LIN {X 0,Y 573.858,Z 220.468,A -85,B 0,C 180,E1 -2228.443,E2 -2228.443} C_VEL
LIN {X 0,Y 573.667,Z 239.844,A -85,B 0,C 180,E1 -2231.425,E2 -2231.425} C_VEL
LIN {X 0,Y 573.432,Z 259.15,A -85,B 0,C 180,E1 -2234.357,E2 -2234.357} C_VEL
LIN {X 0,Y 573.37,Z 271.275,A -85,B 0,C 180,E1 -2236.148,E2 -2236.148} C_VEL
LIN {X 0,Y 574.08,Z 276.429,A -85,B 0,C 180,E1 -2236.256,E2 -2236.256} C_VEL
LIN {X 0,Y 573.913,Z 378.895,A -85,B 0,C 180,E1 -2237.557,E2 -2237.557} C_VEL
LIN {X 0,Y 573.795,Z 392.184,A -85,B 0,C 180,E1 -2237.869,E2 -2237.869} C_VEL
LIN {X 0,Y 573.682,Z 404.351,A -85,B 0,C 180,E1 -2238.293,E2 -2238.293} C_VEL
LIN {X 0,Y 573.582,Z 416.727,A -85,B 0,C 180,E1 -2238.879,E2 -2238.879} C_VEL
LIN {X 0,Y 573.432,Z 428.185,A -85,B 0,C 180,E1 -2239.584,E2 -2239.584} C_VEL
LIN {X 0,Y 573.329,Z 438.59,A -85,B 0,C 180,E1 -2240.384,E2 -2240.384} C_VEL
LIN {X 0,Y 573.238,Z 447.066,A -85,B 0,C 180,E1 -2241.184,E2 -2241.184} C_VEL
LIN {X 0,Y 573.162,Z 454.952,A -85,B 0,C 180,E1 -2242.07,E2 -2242.07} C_VEL
LIN {X 0,Y 573.077,Z 462.942,A -85,B 0,C 180,E1 -2243.183,E2 -2243.183} C_VEL
LIN {X 0,Y 573.071,Z 469.674,A -85,B 0,C 180,E1 -2244.369,E2 -2244.369} C_VEL
LIN {X 0,Y 573.029,Z 474.368,A -85,B 0,C 180,E1 -2245.426,E2 -2245.426} C_VEL
LIN {X 0,Y 573.023,Z 477.954,A -85,B 0,C 180,E1 -2246.483,E2 -2246.483} C_VEL
LIN {X 0,Y 572.959,Z 479.805,A -85,B 0,C 180,E1 -2247.187,E2 -2247.187} C_VEL
LIN {X 0,Y 572.946,Z 482.184,A -85,B 0,C 180,E1 -2248.593,E2 -2248.593} C_VEL
LIN {X 0,Y 572.938,Z 483,A -85,B 0,C 180,E1 -2249.999,E2 -2249.999} C_VEL
LIN {X 0,Y 572.946,Z 482.187,A -85,B 0,C 180,E1 -2251.405,E2 -2251.405} C_VEL
LIN {X 0,Y 572.959,Z 479.813,A -85,B 0,C 180,E1 -2252.811,E2 -2252.811} C_VEL
LIN {X 0,Y 573.014,Z 476.899,A -85,B 0,C 180,E1 -2253.867,E2 -2253.867} C_VEL
LIN {X 0,Y 572.963,Z 472.953,A -85,B 0,C 180,E1 -2254.924,E2 -2254.924} C_VEL
LIN {X 0,Y 573.093,Z 467.873,A -85,B 0,C 180,E1 -2255.982,E2 -2255.982} C_VEL
LIN {X 0,Y 573.083,Z 461.476,A -85,B 0,C 180,E1 -2257.043,E2 -2257.043} C_VEL
LIN {X 0,Y 573.175,Z 453.488,A -85,B 0,C 180,E1 -2258.105,E2 -2258.105} C_VEL
LIN {X 0,Y 573.286,Z 443.551,A -85,B 0,C 180,E1 -2259.169,E2 -2259.169} C_VEL
LIN {X 0,Y 573.409,Z 433.113,A -85,B 0,C 180,E1 -2260.057,E2 -2260.057} C_VEL
LIN {X 0,Y 573.553,Z 421.372,A -85,B 0,C 180,E1 -2260.856,E2 -2260.856} C_VEL
LIN {X 0,Y 573.653,Z 410.31,A -85,B 0,C 180,E1 -2261.446,E2 -2261.446} C_VEL
LIN {X 0,Y 573.757,Z 397.206,A -85,B 0,C 180,E1 -2261.973,E2 -2261.973} C_VEL
LIN {X 0,Y 573.859,Z 384.568,A -85,B 0,C 180,E1 -2262.33,E2 -2262.33} C_VEL
LIN {X 0,Y 573.898,Z 371.408,A -85,B 0,C 180,E1 -2262.553,E2 -2262.553} C_VEL
LIN {X 0,Y 574.043,Z 275.713,A -85,B 0,C 180,E1 -2263.754,E2 -2263.754} C_VEL
LIN {X 0,Y 573.377,Z 271.322,A -85,B 0,C 180,E1 -2263.85,E2 -2263.85} C_VEL
LIN {X 0,Y 573.466,Z 255.545,A -85,B 0,C 180,E1 -2266.188,E2 -2266.188} C_VEL
LIN {X 0,Y 573.648,Z 238.652,A -85,B 0,C 180,E1 -2268.758,E2 -2268.758} C_VEL
LIN {X 0,Y 573.886,Z 220.44,A -85,B 0,C 180,E1 -2271.553,E2 -2271.553} C_VEL
LIN {X 0,Y 573.29,Z 215.695,A -85,B 0,C 180,E1 -2272.334,E2 -2272.334} C_VEL
LIN {X 0,Y 573.248,Z 215.58,A -85,B 0,C 180,E1 -2275.409,E2 -2275.409} C_VEL
LIN {X 0,Y 573.25,Z 215.579,A -85,B 0,C 180,E1 -2278.027,E2 -2278.027} C_VEL
LIN {X 0,Y 573.227,Z 215.575,A -85,B 0,C 180,E1 -2280.88,E2 -2280.88} C_VEL
LIN {X 0,Y 573.263,Z 215.574,A -85,B 0,C 180,E1 -2283.522,E2 -2283.522} C_VEL
LIN {X 0,Y 573.191,Z 215.59,A -85,B 0,C 180,E1 -2286.051,E2 -2286.051} C_VEL
LIN {X 0,Y 573.235,Z 215.575,A -85,B 0,C 180,E1 -2288.7,E2 -2288.7} C_VEL
LIN {X 0,Y 573.224,Z 215.577,A -85,B 0,C 180,E1 -2291.591,E2 -2291.591} C_VEL
LIN {X 0,Y 573.219,Z 215.585,A -85,B 0,C 180,E1 -2294.333,E2 -2294.333} C_VEL
LIN {X 0,Y 573.229,Z 215.573,A -85,B 0,C 180,E1 -2297.358,E2 -2297.358} C_VEL
LIN {X 0,Y 573.232,Z 215.585,A -85,B 0,C 180,E1 -2300.39,E2 -2300.39} C_VEL
LIN {X 0,Y 573.225,Z 215.577,A -85,B 0,C 180,E1 -2303.074,E2 -2303.074} C_VEL
LIN {X 0,Y 573.256,Z 215.571,A -85,B 0,C 180,E1 -2305.669,E2 -2305.669} C_VEL
LIN {X 0,Y 573.23,Z 215.577,A -85,B 0,C 180,E1 -2308.182,E2 -2308.182} C_VEL
LIN {X 0,Y 573.234,Z 215.584,A -85,B 0,C 180,E1 -2310.631,E2 -2310.631} C_VEL
LIN {X 0,Y 573.204,Z 215.578,A -85,B 0,C 180,E1 -2313.511,E2 -2313.511} C_VEL
LIN {X 0,Y 573.19,Z 215.58,A -85,B 0,C 180,E1 -2316.131,E2 -2316.131} C_VEL
LIN {X 0,Y 573.243,Z 215.579,A -85,B 0,C 180,E1 -2318.707,E2 -2318.707} C_VEL
LIN {X 0,Y 573.196,Z 215.583,A -85,B 0,C 180,E1 -2321.408,E2 -2321.408} C_VEL
LIN {X 0,Y 573.216,Z 215.578,A -85,B 0,C 180,E1 -2323.619,E2 -2323.619} C_VEL
LIN {X 0,Y 573.194,Z 215.581,A -85,B 0,C 180,E1 -2326.526,E2 -2326.526} C_VEL
LIN {X 0,Y 573.23,Z 215.582,A -85,B 0,C 180,E1 -2329.4,E2 -2329.4} C_VEL
LIN {X 0,Y 573.198,Z 215.577,A -85,B 0,C 180,E1 -2332.246,E2 -2332.246} C_VEL
LIN {X 0,Y 573.243,Z 215.573,A -85,B 0,C 180,E1 -2334.369,E2 -2334.369} C_VEL
LIN {X 0,Y 573.282,Z 215.573,A -85,B 0,C 180,E1 -2337.187,E2 -2337.187} C_VEL
LIN {X 0,Y 573.28,Z 215.571,A -85,B 0,C 180,E1 -2339.997,E2 -2339.997} C_VEL
LIN {X 0,Y 573.256,Z 215.572,A -85,B 0,C 180,E1 -2342.808,E2 -2342.808} C_VEL
LIN {X 0,Y 573.253,Z 215.581,A -85,B 0,C 180,E1 -2345.626,E2 -2345.626} C_VEL
LIN {X 0,Y 573.224,Z 215.576,A -85,B 0,C 180,E1 -2348.457,E2 -2348.457} C_VEL
LIN {X 0,Y 573.251,Z 215.574,A -85,B 0,C 180,E1 -2351.309,E2 -2351.309} C_VEL
LIN {X 0,Y 573.246,Z 215.576,A -85,B 0,C 180,E1 -2354.416,E2 -2354.416} C_VEL
LIN {X 0,Y 573.222,Z 215.575,A -85,B 0,C 180,E1 -2357.109,E2 -2357.109} C_VEL
LIN {X 0,Y 573.215,Z 215.587,A -85,B 0,C 180,E1 -2360.074,E2 -2360.074} C_VEL
LIN {X 0,Y 573.212,Z 215.584,A -85,B 0,C 180,E1 -2362.335,E2 -2362.335} C_VEL
LIN {X 0,Y 573.216,Z 215.579,A -85,B 0,C 180,E1 -2364.339,E2 -2364.339} C_VEL
LIN {X 0,Y 572.584,Z 215.658,A -85,B 0,C 180,E1 -2364.925,E2 -2364.925} C_VEL
LIN {X 0,Y 569.731,Z 216.014,A -85,B 0,C 180,E1 -2365.876,E2 -2365.876} C_VEL
LIN {X 0,Y 567.297,Z 216.318,A -85,B 0,C 180,E1 -2366.642,E2 -2366.642} C_VEL
LIN {X 0,Y 566.25,Z 216.444,A -85,B 0,C 180,E1 -2367.233,E2 -2367.233} C_VEL
LIN {X 0,Y 566.166,Z 216.455,A -85,B 0,C 180,E1 -2367.433,E2 -2367.433} C_VEL
LIN {X 0,Y 566.171,Z 216.455,A -85,B 0,C 180,E1 -2369.766,E2 -2369.766} C_VEL
LIN {X 0,Y 566.176,Z 216.462,A -85,B 0,C 180,E1 -2372.428,E2 -2372.428} C_VEL
LIN {X 0,Y 566.183,Z 216.455,A -85,B 0,C 180,E1 -2374.992,E2 -2374.992} C_VEL
LIN {X 0,Y 566.163,Z 216.456,A -85,B 0,C 180,E1 -2377.458,E2 -2377.458} C_VEL
LIN {X 0,Y 566.192,Z 216.456,A -85,B 0,C 180,E1 -2380.195,E2 -2380.195} C_VEL
LIN {X 0,Y 566.173,Z 216.46,A -85,B 0,C 180,E1 -2383.051,E2 -2383.051} C_VEL
LIN {X 0,Y 566.164,Z 216.457,A -85,B 0,C 180,E1 -2386.046,E2 -2386.046} C_VEL
LIN {X 0,Y 566.219,Z 216.558,A -85,B 0,C 180,E1 -2388.274,E2 -2388.274} C_VEL
LIN {X 0,Y 566.643,Z 221.534,A -85,B 0,C 180,E1 -2389.156,E2 -2389.156} C_VEL
LIN {X 0,Y 566.439,Z 237.949,A -85,B 0,C 180,E1 -2391.885,E2 -2391.885} C_VEL
LIN {X 0,Y 566.258,Z 253.581,A -85,B 0,C 180,E1 -2394.502,E2 -2394.502} C_VEL
LIN {X 0,Y 566.297,Z 256.947,A -85,B 0,C 180,E1 -2395.023,E2 -2395.023} C_VEL
LIN {X 0,Y 567.157,Z 262.973,A -85,B 0,C 180,E1 -2395.149,E2 -2395.149} C_VEL
LIN {X 0,Y 566.966,Z 364.406,A -85,B 0,C 180,E1 -2396.457,E2 -2396.457} C_VEL
LIN {X 0,Y 566.839,Z 377.799,A -85,B 0,C 180,E1 -2396.781,E2 -2396.781} C_VEL
LIN {X 0,Y 566.728,Z 390.782,A -85,B 0,C 180,E1 -2397.251,E2 -2397.251} C_VEL
LIN {X 0,Y 566.569,Z 403.25,A -85,B 0,C 180,E1 -2397.872,E2 -2397.872} C_VEL
LIN {X 0,Y 566.396,Z 414.525,A -85,B 0,C 180,E1 -2398.592,E2 -2398.592} C_VEL
LIN {X 0,Y 566.301,Z 424.819,A -85,B 0,C 180,E1 -2399.416,E2 -2399.416} C_VEL
LIN {X 0,Y 566.21,Z 433.951,A -85,B 0,C 180,E1 -2400.317,E2 -2400.317} C_VEL
LIN {X 0,Y 566.073,Z 443.236,A -85,B 0,C 180,E1 -2401.448,E2 -2401.448} C_VEL
LIN {X 0,Y 565.988,Z 449.854,A -85,B 0,C 180,E1 -2402.45,E2 -2402.45} C_VEL
LIN {X 0,Y 565.969,Z 455.204,A -85,B 0,C 180,E1 -2403.448,E2 -2403.448} C_VEL
LIN {X 0,Y 565.912,Z 460.191,A -85,B 0,C 180,E1 -2404.632,E2 -2404.632} C_VEL
LIN {X 0,Y 565.854,Z 463.836,A -85,B 0,C 180,E1 -2405.805,E2 -2405.805} C_VEL
LIN {X 0,Y 565.84,Z 465.998,A -85,B 0,C 180,E1 -2406.785,E2 -2406.785} C_VEL
LIN {X 0,Y 565.815,Z 467.646,A -85,B 0,C 180,E1 -2408.123,E2 -2408.123} C_VEL
LIN {X 0,Y 565.863,Z 467.972,A -85,B 0,C 180,E1 -2408.89,E2 -2408.89} C_VEL
LIN {X 0,Y 565.845,Z 467.854,A -85,B 0,C 180,E1 -2409.65,E2 -2409.65} C_VEL
LIN {X 0,Y 565.851,Z 466.913,A -85,B 0,C 180,E1 -2410.709,E2 -2410.709} C_VEL
LIN {X 0,Y 565.866,Z 464.762,A -85,B 0,C 180,E1 -2411.912,E2 -2411.912} C_VEL
LIN {X 0,Y 565.887,Z 461.833,A -85,B 0,C 180,E1 -2412.982,E2 -2412.982} C_VEL
LIN {X 0,Y 565.927,Z 457.463,A -85,B 0,C 180,E1 -2414.146,E2 -2414.146} C_VEL
LIN {X 0,Y 565.991,Z 451.828,A -85,B 0,C 180,E1 -2415.291,E2 -2415.291} C_VEL
LIN {X 0,Y 566.045,Z 445.238,A -85,B 0,C 180,E1 -2416.356,E2 -2416.356} C_VEL
LIN {X 0,Y 566.121,Z 436.817,A -85,B 0,C 180,E1 -2417.454,E2 -2417.454} C_VEL
LIN {X 0,Y 566.231,Z 428.168,A -85,B 0,C 180,E1 -2418.365,E2 -2418.365} C_VEL
LIN {X 0,Y 566.398,Z 417.508,A -85,B 0,C 180,E1 -2419.275,E2 -2419.275} C_VEL
LIN {X 0,Y 566.501,Z 406.986,A -85,B 0,C 180,E1 -2419.999,E2 -2419.999} C_VEL
LIN {X 0,Y 566.685,Z 395.322,A -85,B 0,C 180,E1 -2420.633,E2 -2420.633} C_VEL
LIN {X 0,Y 566.818,Z 383.255,A -85,B 0,C 180,E1 -2421.13,E2 -2421.13} C_VEL
LIN {X 0,Y 566.909,Z 370.18,A -85,B 0,C 180,E1 -2421.513,E2 -2421.513} C_VEL
LIN {X 0,Y 566.986,Z 357.597,A -85,B 0,C 180,E1 -2421.739,E2 -2421.739} C_VEL
LIN {X 0,Y 567.011,Z 261.658,A -85,B 0,C 180,E1 -2422.961,E2 -2422.961} C_VEL
LIN {X 0,Y 566.311,Z 256.974,A -85,B 0,C 180,E1 -2423.065,E2 -2423.065} C_VEL
LIN {X 0,Y 566.369,Z 245.017,A -85,B 0,C 180,E1 -2425.018,E2 -2425.018} C_VEL
LIN {X 0,Y 566.537,Z 230.243,A -85,B 0,C 180,E1 -2427.513,E2 -2427.513} C_VEL
LIN {X 0,Y 566.602,Z 218.801,A -85,B 0,C 180,E1 -2429.468,E2 -2429.468} C_VEL
LIN {X 0,Y 566.238,Z 216.532,A -85,B 0,C 180,E1 -2429.912,E2 -2429.912} C_VEL
LIN {X 0,Y 566.234,Z 216.451,A -85,B 0,C 180,E1 -2432.847,E2 -2432.847} C_VEL
LIN {X 0,Y 566.226,Z 216.453,A -85,B 0,C 180,E1 -2435.7,E2 -2435.7} C_VEL
LIN {X 0,Y 566.184,Z 216.452,A -85,B 0,C 180,E1 -2438.567,E2 -2438.567} C_VEL
LIN {X 0,Y 566.198,Z 216.459,A -85,B 0,C 180,E1 -2441.456,E2 -2441.456} C_VEL
LIN {X 0,Y 566.179,Z 216.453,A -85,B 0,C 180,E1 -2444.504,E2 -2444.504} C_VEL
LIN {X 0,Y 566.16,Z 216.458,A -85,B 0,C 180,E1 -2447.334,E2 -2447.334} C_VEL
LIN {X 0,Y 566.17,Z 216.457,A -85,B 0,C 180,E1 -2450.34,E2 -2450.34} C_VEL
LIN {X 0,Y 566.131,Z 216.46,A -85,B 0,C 180,E1 -2453.284,E2 -2453.284} C_VEL
LIN {X 0,Y 566.157,Z 216.461,A -85,B 0,C 180,E1 -2455.753,E2 -2455.753} C_VEL
LIN {X 0,Y 566.147,Z 216.457,A -85,B 0,C 180,E1 -2458.957,E2 -2458.957} C_VEL
LIN {X 0,Y 566.158,Z 216.455,A -85,B 0,C 180,E1 -2461.425,E2 -2461.425} C_VEL
LIN {X 0,Y 566.16,Z 216.459,A -85,B 0,C 180,E1 -2463.96,E2 -2463.96} C_VEL
LIN {X 0,Y 566.141,Z 216.465,A -85,B 0,C 180,E1 -2466.575,E2 -2466.575} C_VEL
LIN {X 0,Y 566.178,Z 216.453,A -85,B 0,C 180,E1 -2469.688,E2 -2469.688} C_VEL
LIN {X 0,Y 566.165,Z 216.46,A -85,B 0,C 180,E1 -2472.92,E2 -2472.92} C_VEL
LIN {X 0,Y 566.168,Z 216.455,A -85,B 0,C 180,E1 -2476.053,E2 -2476.053} C_VEL
LIN {X 0,Y 566.179,Z 216.457,A -85,B 0,C 180,E1 -2479.219,E2 -2479.219} C_VEL
LIN {X 0,Y 566.157,Z 216.456,A -85,B 0,C 180,E1 -2481.64,E2 -2481.64} C_VEL
LIN {X 0,Y 566.142,Z 216.458,A -85,B 0,C 180,E1 -2484.311,E2 -2484.311} C_VEL
LIN {X 0,Y 566.177,Z 216.46,A -85,B 0,C 180,E1 -2486.9,E2 -2486.9} C_VEL
LIN {X 0,Y 566.148,Z 216.463,A -85,B 0,C 180,E1 -2489.41,E2 -2489.41} C_VEL
LIN {X 0,Y 566.158,Z 216.457,A -85,B 0,C 180,E1 -2491.859,E2 -2491.859} C_VEL
LIN {X 0,Y 566.161,Z 216.455,A -85,B 0,C 180,E1 -2494.253,E2 -2494.253} C_VEL
LIN {X 0,Y 566.157,Z 216.456,A -85,B 0,C 180,E1 -2496.724,E2 -2496.724} C_VEL
LIN {X 0,Y 566.196,Z 216.458,A -85,B 0,C 180,E1 -2499.666,E2 -2499.666} C_VEL
LIN {X 0,Y 566.165,Z 216.459,A -85,B 0,C 180,E1 -2501.924,E2 -2501.924} C_VEL
LIN {X 0,Y 566.181,Z 216.453,A -85,B 0,C 180,E1 -2504.893,E2 -2504.893} C_VEL
LIN {X 0,Y 566.211,Z 216.459,A -85,B 0,C 180,E1 -2507.822,E2 -2507.822} C_VEL
LIN {X 0,Y 566.185,Z 216.452,A -85,B 0,C 180,E1 -2510.717,E2 -2510.717} C_VEL
LIN {X 0,Y 566.169,Z 216.458,A -85,B 0,C 180,E1 -2513.589,E2 -2513.589} C_VEL
LIN {X 0,Y 566.172,Z 216.459,A -85,B 0,C 180,E1 -2515.732,E2 -2515.732} C_VEL
LIN {X 0,Y 566.276,Z 216.447,A -85,B 0,C 180,E1 -2517.869,E2 -2517.869} C_VEL
LIN {X 0,Y 566.299,Z 216.44,A -85,B 0,C 180,E1 -2520.714,E2 -2520.714} C_VEL
LIN {X 0,Y 566.261,Z 216.444,A -85,B 0,C 180,E1 -2522.848,E2 -2522.848} C_VEL
LIN {X 0,Y 566.234,Z 216.447,A -85,B 0,C 180,E1 -2525.701,E2 -2525.701} C_VEL
LIN {X 0,Y 566.196,Z 216.459,A -85,B 0,C 180,E1 -2528.569,E2 -2528.569} C_VEL
LIN {X 0,Y 566.25,Z 216.444,A -85,B 0,C 180,E1 -2531.456,E2 -2531.456} C_VEL
LIN {X 0,Y 566.222,Z 216.456,A -85,B 0,C 180,E1 -2534.499,E2 -2534.499} C_VEL
LIN {X 0,Y 566.198,Z 216.452,A -85,B 0,C 180,E1 -2537.334,E2 -2537.334} C_VEL
LIN {X 0,Y 566.21,Z 216.449,A -85,B 0,C 180,E1 -2539.583,E2 -2539.583} C_VEL
LIN {X 0,Y 566.196,Z 216.45,A -85,B 0,C 180,E1 -2541.865,E2 -2541.865} C_VEL
LIN {X 0,Y 566.191,Z 216.461,A -85,B 0,C 180,E1 -2545.022,E2 -2545.022} C_VEL
LIN {X 0,Y 566.178,Z 216.458,A -85,B 0,C 180,E1 -2547.343,E2 -2547.343} C_VEL
LIN {X 0,Y 566.18,Z 216.454,A -85,B 0,C 180,E1 -2549.772,E2 -2549.772} C_VEL
LIN {X 0,Y 566.204,Z 216.45,A -85,B 0,C 180,E1 -2552.429,E2 -2552.429} C_VEL
LIN {X 0,Y 566.178,Z 216.458,A -85,B 0,C 180,E1 -2554.988,E2 -2554.988} C_VEL
LIN {X 0,Y 566.203,Z 216.459,A -85,B 0,C 180,E1 -2557.462,E2 -2557.462} C_VEL
LIN {X 0,Y 566.219,Z 216.448,A -85,B 0,C 180,E1 -2560.2,E2 -2560.2} C_VEL
LIN {X 0,Y 566.19,Z 216.454,A -85,B 0,C 180,E1 -2563.057,E2 -2563.057} C_VEL
LIN {X 0,Y 566.168,Z 216.458,A -85,B 0,C 180,E1 -2566.054,E2 -2566.054} C_VEL
LIN {X 0,Y 566.169,Z 216.454,A -85,B 0,C 180,E1 -2568.859,E2 -2568.859} C_VEL
LIN {X 0,Y 566.216,Z 216.452,A -85,B 0,C 180,E1 -2571.443,E2 -2571.443} C_VEL
LIN {X 0,Y 566.153,Z 216.46,A -85,B 0,C 180,E1 -2574.306,E2 -2574.306} C_VEL
LIN {X 0,Y 566.22,Z 216.448,A -85,B 0,C 180,E1 -2576.897,E2 -2576.897} C_VEL
LIN {X 0,Y 566.179,Z 216.454,A -85,B 0,C 180,E1 -2579.406,E2 -2579.406} C_VEL
LIN {X 0,Y 566.199,Z 216.456,A -85,B 0,C 180,E1 -2581.856,E2 -2581.856} C_VEL
LIN {X 0,Y 566.205,Z 216.461,A -85,B 0,C 180,E1 -2584.25,E2 -2584.25} C_VEL
LIN {X 0,Y 566.199,Z 216.458,A -85,B 0,C 180,E1 -2587.368,E2 -2587.368} C_VEL
LIN {X 0,Y 566.262,Z 216.781,A -85,B 0,C 180,E1 -2587.563,E2 -2587.563} C_VEL
LIN {X 0,Y 566.913,Z 221.888,A -85,B 0,C 180,E1 -2588.401,E2 -2588.401} C_VEL
LIN {X 0,Y 566.69,Z 241.013,A -85,B 0,C 180,E1 -2591.376,E2 -2591.376} C_VEL
LIN {X 0,Y 566.443,Z 259.15,A -85,B 0,C 180,E1 -2594.159,E2 -2594.159} C_VEL
LIN {X 0,Y 566.366,Z 271.284,A -85,B 0,C 180,E1 -2595.973,E2 -2595.973} C_VEL
LIN {X 0,Y 567.189,Z 277.032,A -85,B 0,C 180,E1 -2596.093,E2 -2596.093} C_VEL
LIN {X 0,Y 566.99,Z 378.894,A -85,B 0,C 180,E1 -2597.403,E2 -2597.403} C_VEL
LIN {X 0,Y 566.863,Z 392.183,A -85,B 0,C 180,E1 -2597.718,E2 -2597.718} C_VEL
LIN {X 0,Y 566.73,Z 404.352,A -85,B 0,C 180,E1 -2598.147,E2 -2598.147} C_VEL
LIN {X 0,Y 566.632,Z 416.137,A -85,B 0,C 180,E1 -2598.707,E2 -2598.707} C_VEL
LIN {X 0,Y 566.447,Z 428.182,A -85,B 0,C 180,E1 -2599.454,E2 -2599.454} C_VEL
LIN {X 0,Y 566.321,Z 438.591,A -85,B 0,C 180,E1 -2600.264,E2 -2600.264} C_VEL
LIN {X 0,Y 566.207,Z 447.081,A -85,B 0,C 180,E1 -2601.073,E2 -2601.073} C_VEL
LIN {X 0,Y 566.113,Z 454.952,A -85,B 0,C 180,E1 -2601.971,E2 -2601.971} C_VEL
LIN {X 0,Y 565.999,Z 462.616,A -85,B 0,C 180,E1 -2603.046,E2 -2603.046} C_VEL
LIN {X 0,Y 566.004,Z 469.674,A -85,B 0,C 180,E1 -2604.298,E2 -2604.298} C_VEL
LIN {X 0,Y 565.933,Z 474.368,A -85,B 0,C 180,E1 -2605.369,E2 -2605.369} C_VEL
LIN {X 0,Y 565.927,Z 477.955,A -85,B 0,C 180,E1 -2606.439,E2 -2606.439} C_VEL
LIN {X 0,Y 565.878,Z 479.805,A -85,B 0,C 180,E1 -2607.151,E2 -2607.151} C_VEL
LIN {X 0,Y 565.845,Z 482.183,A -85,B 0,C 180,E1 -2608.575,E2 -2608.575} C_VEL
LIN {X 0,Y 565.839,Z 483,A -85,B 0,C 180,E1 -2609.999,E2 -2609.999} C_VEL
LIN {X 0,Y 565.845,Z 482.187,A -85,B 0,C 180,E1 -2611.422,E2 -2611.422} C_VEL
LIN {X 0,Y 565.878,Z 479.813,A -85,B 0,C 180,E1 -2612.846,E2 -2612.846} C_VEL
LIN {X 0,Y 565.926,Z 476.899,A -85,B 0,C 180,E1 -2613.915,E2 -2613.915} C_VEL
LIN {X 0,Y 565.878,Z 472.953,A -85,B 0,C 180,E1 -2614.986,E2 -2614.986} C_VEL
LIN {X 0,Y 566.006,Z 467.873,A -85,B 0,C 180,E1 -2616.057,E2 -2616.057} C_VEL
LIN {X 0,Y 566.033,Z 461.476,A -85,B 0,C 180,E1 -2617.131,E2 -2617.131} C_VEL
LIN {X 0,Y 566.129,Z 453.488,A -85,B 0,C 180,E1 -2618.207,E2 -2618.207} C_VEL
LIN {X 0,Y 566.229,Z 445.346,A -85,B 0,C 180,E1 -2619.104,E2 -2619.104} C_VEL
LIN {X 0,Y 566.332,Z 435.414,A -85,B 0,C 180,E1 -2620.004,E2 -2620.004} C_VEL
LIN {X 0,Y 566.547,Z 424.304,A -85,B 0,C 180,E1 -2620.806,E2 -2620.806} C_VEL
LIN {X 0,Y 566.661,Z 413.198,A -85,B 0,C 180,E1 -2621.444,E2 -2621.444} C_VEL
LIN {X 0,Y 566.746,Z 401.011,A -85,B 0,C 180,E1 -2621.987,E2 -2621.987} C_VEL
LIN {X 0,Y 566.911,Z 388.225,A -85,B 0,C 180,E1 -2622.392,E2 -2622.392} C_VEL
LIN {X 0,Y 566.995,Z 374.683,A -85,B 0,C 180,E1 -2622.663,E2 -2622.663} C_VEL
LIN {X 0,Y 567.039,Z 275.928,A -85,B 0,C 180,E1 -2623.925,E2 -2623.925} C_VEL
LIN {X 0,Y 566.371,Z 271.333,A -85,B 0,C 180,E1 -2624.025,E2 -2624.025} C_VEL
LIN {X 0,Y 566.47,Z 257.958,A -85,B 0,C 180,E1 -2626.023,E2 -2626.023} C_VEL
LIN {X 0,Y 566.687,Z 241.01,A -85,B 0,C 180,E1 -2628.622,E2 -2628.622} C_VEL
LIN {X 0,Y 566.923,Z 221.779,A -85,B 0,C 180,E1 -2631.602,E2 -2631.602} C_VEL
LIN {X 0,Y 566.229,Z 216.528,A -85,B 0,C 180,E1 -2632.484,E2 -2632.484} C_VEL
LIN {X 0,Y 566.212,Z 216.459,A -85,B 0,C 180,E1 -2635.748,E2 -2635.748} C_VEL
LIN {X 0,Y 566.204,Z 216.454,A -85,B 0,C 180,E1 -2638.2,E2 -2638.2} C_VEL
LIN {X 0,Y 566.191,Z 216.452,A -85,B 0,C 180,E1 -2641.075,E2 -2641.075} C_VEL
LIN {X 0,Y 566.211,Z 216.456,A -85,B 0,C 180,E1 -2643.732,E2 -2643.732} C_VEL
LIN {X 0,Y 566.18,Z 216.456,A -85,B 0,C 180,E1 -2646.57,E2 -2646.57} C_VEL
LIN {X 0,Y 566.211,Z 216.452,A -85,B 0,C 180,E1 -2649.684,E2 -2649.684} C_VEL
LIN {X 0,Y 566.194,Z 216.452,A -85,B 0,C 180,E1 -2652.915,E2 -2652.915} C_VEL
LIN {X 0,Y 566.19,Z 216.458,A -85,B 0,C 180,E1 -2656.048,E2 -2656.048} C_VEL
LIN {X 0,Y 566.2,Z 216.451,A -85,B 0,C 180,E1 -2659.213,E2 -2659.213} C_VEL
LIN {X 0,Y 566.176,Z 216.454,A -85,B 0,C 180,E1 -2661.634,E2 -2661.634} C_VEL
LIN {X 0,Y 566.144,Z 216.464,A -85,B 0,C 180,E1 -2664.305,E2 -2664.305} C_VEL
LIN {X 0,Y 566.205,Z 216.455,A -85,B 0,C 180,E1 -2666.895,E2 -2666.895} C_VEL
LIN {X 0,Y 566.162,Z 216.456,A -85,B 0,C 180,E1 -2669.404,E2 -2669.404} C_VEL
LIN {X 0,Y 566.181,Z 216.452,A -85,B 0,C 180,E1 -2671.854,E2 -2671.854} C_VEL
LIN {X 0,Y 566.184,Z 216.454,A -85,B 0,C 180,E1 -2674.248,E2 -2674.248} C_VEL
LIN {X 0,Y 566.154,Z 216.459,A -85,B 0,C 180,E1 -2677.365,E2 -2677.365} C_VEL
LIN {X 0,Y 566.191,Z 216.452,A -85,B 0,C 180,E1 -2679.66,E2 -2679.66} C_VEL
LIN {X 0,Y 566.167,Z 216.454,A -85,B 0,C 180,E1 -2681.919,E2 -2681.919} C_VEL
LIN {X 0,Y 566.173,Z 216.46,A -85,B 0,C 180,E1 -2684.888,E2 -2684.888} C_VEL
LIN {X 0,Y 566.166,Z 216.455,A -85,B 0,C 180,E1 -2687.815,E2 -2687.815} C_VEL
LIN {X 0,Y 566.135,Z 216.459,A -85,B 0,C 180,E1 -2689.989,E2 -2689.989} C_VEL
LIN {X 0,Y 566.221,Z 216.449,A -85,B 0,C 180,E1 -2692.868,E2 -2692.868} C_VEL
LIN {X 0,Y 566.258,Z 216.447,A -85,B 0,C 180,E1 -2695.013,E2 -2695.013} C_VEL
LIN {X 0,Y 566.243,Z 216.449,A -85,B 0,C 180,E1 -2697.863,E2 -2697.863} C_VEL
LIN {X 0,Y 566.251,Z 216.446,A -85,B 0,C 180,E1 -2699.997,E2 -2699.997} C_VEL
LIN {X 0,Y 566.226,Z 216.447,A -85,B 0,C 180,E1 -2702.843,E2 -2702.843} C_VEL
LIN {X 0,Y 566.221,Z 216.457,A -85,B 0,C 180,E1 -2705.696,E2 -2705.696} C_VEL
LIN {X 0,Y 566.176,Z 216.453,A -85,B 0,C 180,E1 -2708.563,E2 -2708.563} C_VEL
LIN {X 0,Y 566.218,Z 216.452,A -85,B 0,C 180,E1 -2711.452,E2 -2711.452} C_VEL
LIN {X 0,Y 566.201,Z 216.452,A -85,B 0,C 180,E1 -2714.499,E2 -2714.499} C_VEL
LIN {X 0,Y 566.164,Z 216.455,A -85,B 0,C 180,E1 -2717.329,E2 -2717.329} C_VEL
LIN {X 0,Y 566.181,Z 216.459,A -85,B 0,C 180,E1 -2720.335,E2 -2720.335} C_VEL
LIN {X 0,Y 566.144,Z 216.457,A -85,B 0,C 180,E1 -2723.279,E2 -2723.279} C_VEL
LIN {X 0,Y 566.178,Z 216.455,A -85,B 0,C 180,E1 -2725.747,E2 -2725.747} C_VEL
LIN {X 0,Y 566.166,Z 216.455,A -85,B 0,C 180,E1 -2727.433,E2 -2727.433} C_VEL
LIN {X 0,Y 565.498,Z 216.545,A -85,B 0,C 180,E1 -2728.027,E2 -2728.027} C_VEL
LIN {X 0,Y 562.638,Z 216.9,A -85,B 0,C 180,E1 -2728.991,E2 -2728.991} C_VEL
LIN {X 0,Y 560.223,Z 217.2,A -85,B 0,C 180,E1 -2729.766,E2 -2729.766} C_VEL
LIN {X 0,Y 559.19,Z 217.334,A -85,B 0,C 180,E1 -2730.365,E2 -2730.365} C_VEL
LIN {X 0,Y 559.109,Z 217.336,A -85,B 0,C 180,E1 -2730.568,E2 -2730.568} C_VEL
LIN {X 0,Y 559.144,Z 217.335,A -85,B 0,C 180,E1 -2732.711,E2 -2732.711} C_VEL
LIN {X 0,Y 559.127,Z 217.331,A -85,B 0,C 180,E1 -2735.319,E2 -2735.319} C_VEL
LIN {X 0,Y 559.102,Z 217.337,A -85,B 0,C 180,E1 -2738.015,E2 -2738.015} C_VEL
LIN {X 0,Y 559.144,Z 217.339,A -85,B 0,C 180,E1 -2740.808,E2 -2740.808} C_VEL
LIN {X 0,Y 559.126,Z 217.333,A -85,B 0,C 180,E1 -2743.729,E2 -2743.729} C_VEL
LIN {X 0,Y 559.135,Z 217.341,A -85,B 0,C 180,E1 -2746.798,E2 -2746.798} C_VEL
LIN {X 0,Y 559.179,Z 217.428,A -85,B 0,C 180,E1 -2748.186,E2 -2748.186} C_VEL
LIN {X 0,Y 559.643,Z 222.307,A -85,B 0,C 180,E1 -2749.059,E2 -2749.059} C_VEL
LIN {X 0,Y 559.422,Z 238.602,A -85,B 0,C 180,E1 -2751.789,E2 -2751.789} C_VEL
LIN {X 0,Y 559.233,Z 254.468,A -85,B 0,C 180,E1 -2754.464,E2 -2754.464} C_VEL
LIN {X 0,Y 559.267,Z 257.004,A -85,B 0,C 180,E1 -2754.848,E2 -2754.848} C_VEL
LIN {X 0,Y 560.262,Z 264.287,A -85,B 0,C 180,E1 -2754.992,E2 -2754.992} C_VEL
LIN {X 0,Y 560.056,Z 364.634,A -85,B 0,C 180,E1 -2756.304,E2 -2756.304} C_VEL
LIN {X 0,Y 559.907,Z 378.199,A -85,B 0,C 180,E1 -2756.639,E2 -2756.639} C_VEL
LIN {X 0,Y 559.77,Z 391.034,A -85,B 0,C 180,E1 -2757.113,E2 -2757.113} C_VEL
LIN {X 0,Y 559.59,Z 403.438,A -85,B 0,C 180,E1 -2757.741,E2 -2757.741} C_VEL
LIN {X 0,Y 559.407,Z 414.453,A -85,B 0,C 180,E1 -2758.455,E2 -2758.455} C_VEL
LIN {X 0,Y 559.275,Z 424.928,A -85,B 0,C 180,E1 -2759.304,E2 -2759.304} C_VEL
LIN {X 0,Y 559.156,Z 434.886,A -85,B 0,C 180,E1 -2760.311,E2 -2760.311} C_VEL
LIN {X 0,Y 559.017,Z 442.545,A -85,B 0,C 180,E1 -2761.259,E2 -2761.259} C_VEL
LIN {X 0,Y 558.914,Z 449.296,A -85,B 0,C 180,E1 -2762.275,E2 -2762.275} C_VEL
LIN {X 0,Y 558.891,Z 454.416,A -85,B 0,C 180,E1 -2763.219,E2 -2763.219} C_VEL
LIN {X 0,Y 558.841,Z 459.103,A -85,B 0,C 180,E1 -2764.288,E2 -2764.288} C_VEL
LIN {X 0,Y 558.811,Z 463.079,A -85,B 0,C 180,E1 -2765.48,E2 -2765.48} C_VEL
LIN {X 0,Y 558.755,Z 465.799,A -85,B 0,C 180,E1 -2766.651,E2 -2766.651} C_VEL
LIN {X 0,Y 558.724,Z 467.434,A -85,B 0,C 180,E1 -2767.831,E2 -2767.831} C_VEL
LIN {X 0,Y 558.753,Z 467.91,A -85,B 0,C 180,E1 -2768.608,E2 -2768.608} C_VEL
LIN {X 0,Y 558.743,Z 467.933,A -85,B 0,C 180,E1 -2769.38,E2 -2769.38} C_VEL
LIN {X 0,Y 558.768,Z 467.054,A -85,B 0,C 180,E1 -2770.603,E2 -2770.603} C_VEL
LIN {X 0,Y 558.75,Z 465.328,A -85,B 0,C 180,E1 -2771.674,E2 -2771.674} C_VEL
LIN {X 0,Y 558.806,Z 462.247,A -85,B 0,C 180,E1 -2772.892,E2 -2772.892} C_VEL
LIN {X 0,Y 558.824,Z 458.565,A -85,B 0,C 180,E1 -2773.939,E2 -2773.939} C_VEL
LIN {X 0,Y 558.889,Z 453.462,A -85,B 0,C 180,E1 -2775.063,E2 -2775.063} C_VEL
LIN {X 0,Y 558.969,Z 447.043,A -85,B 0,C 180,E1 -2776.18,E2 -2776.18} C_VEL
LIN {X 0,Y 559.067,Z 439.003,A -85,B 0,C 180,E1 -2777.293,E2 -2777.293} C_VEL
LIN {X 0,Y 559.162,Z 430.826,A -85,B 0,C 180,E1 -2778.216,E2 -2778.216} C_VEL
LIN {X 0,Y 559.336,Z 420.857,A -85,B 0,C 180,E1 -2779.138,E2 -2779.138} C_VEL
LIN {X 0,Y 559.518,Z 409.673,A -85,B 0,C 180,E1 -2779.964,E2 -2779.964} C_VEL
LIN {X 0,Y 559.68,Z 398.736,A -85,B 0,C 180,E1 -2780.606,E2 -2780.606} C_VEL
LIN {X 0,Y 559.845,Z 386.674,A -85,B 0,C 180,E1 -2781.155,E2 -2781.155} C_VEL
LIN {X 0,Y 559.977,Z 374.28,A -85,B 0,C 180,E1 -2781.566,E2 -2781.566} C_VEL
LIN {X 0,Y 560.068,Z 361.452,A -85,B 0,C 180,E1 -2781.84,E2 -2781.84} C_VEL
LIN {X 0,Y 560.113,Z 262.225,A -85,B 0,C 180,E1 -2783.129,E2 -2783.129} C_VEL
LIN {X 0,Y 559.266,Z 257.027,A -85,B 0,C 180,E1 -2783.242,E2 -2783.242} C_VEL
LIN {X 0,Y 559.321,Z 249.81,A -85,B 0,C 180,E1 -2784.413,E2 -2784.413} C_VEL
LIN {X 0,Y 559.549,Z 232.883,A -85,B 0,C 180,E1 -2787.301,E2 -2787.301} C_VEL
LIN {X 0,Y 559.669,Z 220.375,A -85,B 0,C 180,E1 -2789.462,E2 -2789.462} C_VEL
LIN {X 0,Y 559.206,Z 217.387,A -85,B 0,C 180,E1 -2790.046,E2 -2790.046} C_VEL
LIN {X 0,Y 559.201,Z 217.328,A -85,B 0,C 180,E1 -2792.883,E2 -2792.883} C_VEL
LIN {X 0,Y 559.193,Z 217.329,A -85,B 0,C 180,E1 -2795.772,E2 -2795.772} C_VEL
LIN {X 0,Y 559.143,Z 217.329,A -85,B 0,C 180,E1 -2798.676,E2 -2798.676} C_VEL
LIN {X 0,Y 559.161,Z 217.338,A -85,B 0,C 180,E1 -2801.602,E2 -2801.602} C_VEL
LIN {X 0,Y 559.137,Z 217.33,A -85,B 0,C 180,E1 -2804.59,E2 -2804.59} C_VEL
LIN {X 0,Y 559.119,Z 217.339,A -85,B 0,C 180,E1 -2807.559,E2 -2807.559} C_VEL
LIN {X 0,Y 559.128,Z 217.342,A -85,B 0,C 180,E1 -2809.84,E2 -2809.84} C_VEL
LIN {X 0,Y 559.1,Z 217.341,A -85,B 0,C 180,E1 -2812.156,E2 -2812.156} C_VEL
LIN {X 0,Y 559.122,Z 217.332,A -85,B 0,C 180,E1 -2815.186,E2 -2815.186} C_VEL
LIN {X 0,Y 559.097,Z 217.341,A -85,B 0,C 180,E1 -2818.378,E2 -2818.378} C_VEL
LIN {X 0,Y 559.111,Z 217.333,A -85,B 0,C 180,E1 -2821.276,E2 -2821.276} C_VEL
LIN {X 0,Y 559.118,Z 217.336,A -85,B 0,C 180,E1 -2823.95,E2 -2823.95} C_VEL
LIN {X 0,Y 559.091,Z 217.337,A -85,B 0,C 180,E1 -2827.113,E2 -2827.113} C_VEL
LIN {X 0,Y 559.126,Z 217.333,A -85,B 0,C 180,E1 -2829.945,E2 -2829.945} C_VEL
LIN {X 0,Y 559.122,Z 217.34,A -85,B 0,C 180,E1 -2832.748,E2 -2832.748} C_VEL
LIN {X 0,Y 559.122,Z 217.332,A -85,B 0,C 180,E1 -2835.765,E2 -2835.765} C_VEL
LIN {X 0,Y 559.101,Z 217.336,A -85,B 0,C 180,E1 -2838.23,E2 -2838.23} C_VEL
LIN {X 0,Y 559.149,Z 217.334,A -85,B 0,C 180,E1 -2841.196,E2 -2841.196} C_VEL
LIN {X 0,Y 559.119,Z 217.332,A -85,B 0,C 180,E1 -2843.793,E2 -2843.793} C_VEL
LIN {X 0,Y 559.128,Z 217.332,A -85,B 0,C 180,E1 -2846.428,E2 -2846.428} C_VEL
LIN {X 0,Y 559.131,Z 217.338,A -85,B 0,C 180,E1 -2848.984,E2 -2848.984} C_VEL
LIN {X 0,Y 559.102,Z 217.338,A -85,B 0,C 180,E1 -2851.633,E2 -2851.633} C_VEL
LIN {X 0,Y 559.11,Z 217.335,A -85,B 0,C 180,E1 -2854.703,E2 -2854.703} C_VEL
LIN {X 0,Y 559.109,Z 217.338,A -85,B 0,C 180,E1 -2857.07,E2 -2857.07} C_VEL
LIN {X 0,Y 559.167,Z 217.335,A -85,B 0,C 180,E1 -2859.399,E2 -2859.399} C_VEL
LIN {X 0,Y 559.117,Z 217.341,A -85,B 0,C 180,E1 -2861.688,E2 -2861.688} C_VEL
LIN {X 0,Y 559.132,Z 217.336,A -85,B 0,C 180,E1 -2863.95,E2 -2863.95} C_VEL
LIN {X 0,Y 559.152,Z 217.331,A -85,B 0,C 180,E1 -2866.187,E2 -2866.187} C_VEL
LIN {X 0,Y 559.164,Z 217.328,A -85,B 0,C 180,E1 -2869.136,E2 -2869.136} C_VEL
LIN {X 0,Y 559.144,Z 217.337,A -85,B 0,C 180,E1 -2872.056,E2 -2872.056} C_VEL
LIN {X 0,Y 559.23,Z 217.318,A -85,B 0,C 180,E1 -2874.956,E2 -2874.956} C_VEL
LIN {X 0,Y 559.248,Z 217.322,A -85,B 0,C 180,E1 -2877.842,E2 -2877.842} C_VEL
LIN {X 0,Y 559.269,Z 217.316,A -85,B 0,C 180,E1 -2880.723,E2 -2880.723} C_VEL
LIN {X 0,Y 559.226,Z 217.32,A -85,B 0,C 180,E1 -2882.884,E2 -2882.884} C_VEL
LIN {X 0,Y 559.205,Z 217.323,A -85,B 0,C 180,E1 -2885.773,E2 -2885.773} C_VEL
LIN {X 0,Y 559.162,Z 217.333,A -85,B 0,C 180,E1 -2888.677,E2 -2888.677} C_VEL
LIN {X 0,Y 559.211,Z 217.321,A -85,B 0,C 180,E1 -2891.603,E2 -2891.603} C_VEL
LIN {X 0,Y 559.171,Z 217.336,A -85,B 0,C 180,E1 -2894.581,E2 -2894.581} C_VEL
LIN {X 0,Y 559.142,Z 217.329,A -85,B 0,C 180,E1 -2897.56,E2 -2897.56} C_VEL
LIN {X 0,Y 559.173,Z 217.325,A -85,B 0,C 180,E1 -2899.839,E2 -2899.839} C_VEL
LIN {X 0,Y 559.142,Z 217.33,A -85,B 0,C 180,E1 -2902.155,E2 -2902.155} C_VEL
LIN {X 0,Y 559.152,Z 217.335,A -85,B 0,C 180,E1 -2905.179,E2 -2905.179} C_VEL
LIN {X 0,Y 559.12,Z 217.333,A -85,B 0,C 180,E1 -2907.717,E2 -2907.717} C_VEL
LIN {X 0,Y 559.147,Z 217.328,A -85,B 0,C 180,E1 -2910.185,E2 -2910.185} C_VEL
LIN {X 0,Y 559.16,Z 217.33,A -85,B 0,C 180,E1 -2912.717,E2 -2912.717} C_VEL
LIN {X 0,Y 559.129,Z 217.342,A -85,B 0,C 180,E1 -2915.326,E2 -2915.326} C_VEL
LIN {X 0,Y 559.139,Z 217.331,A -85,B 0,C 180,E1 -2918.019,E2 -2918.019} C_VEL
LIN {X 0,Y 559.139,Z 217.331,A -85,B 0,C 180,E1 -2920.816,E2 -2920.816} C_VEL
LIN {X 0,Y 559.119,Z 217.34,A -85,B 0,C 180,E1 -2923.738,E2 -2923.738} C_VEL
LIN {X 0,Y 559.119,Z 217.334,A -85,B 0,C 180,E1 -2926.263,E2 -2926.263} C_VEL
LIN {X 0,Y 559.154,Z 217.328,A -85,B 0,C 180,E1 -2928.952,E2 -2928.952} C_VEL
LIN {X 0,Y 559.182,Z 217.326,A -85,B 0,C 180,E1 -2931.192,E2 -2931.192} C_VEL
LIN {X 0,Y 559.128,Z 217.34,A -85,B 0,C 180,E1 -2933.787,E2 -2933.787} C_VEL
LIN {X 0,Y 559.171,Z 217.329,A -85,B 0,C 180,E1 -2936.425,E2 -2936.425} C_VEL
LIN {X 0,Y 559.159,Z 217.327,A -85,B 0,C 180,E1 -2938.98,E2 -2938.98} C_VEL
LIN {X 0,Y 559.155,Z 217.331,A -85,B 0,C 180,E1 -2941.623,E2 -2941.623} C_VEL
LIN {X 0,Y 559.172,Z 217.332,A -85,B 0,C 180,E1 -2943.902,E2 -2943.902} C_VEL
LIN {X 0,Y 559.134,Z 217.338,A -85,B 0,C 180,E1 -2947.066,E2 -2947.066} C_VEL
LIN {X 0,Y 559.219,Z 217.643,A -85,B 0,C 180,E1 -2947.411,E2 -2947.411} C_VEL
LIN {X 0,Y 559.98,Z 223.326,A -85,B 0,C 180,E1 -2948.361,E2 -2948.361} C_VEL
LIN {X 0,Y 559.692,Z 242.153,A -85,B 0,C 180,E1 -2951.324,E2 -2951.324} C_VEL
LIN {X 0,Y 559.448,Z 259.119,A -85,B 0,C 180,E1 -2953.955,E2 -2953.955} C_VEL
LIN {X 0,Y 559.37,Z 271.293,A -85,B 0,C 180,E1 -2955.794,E2 -2955.794} C_VEL
LIN {X 0,Y 560.303,Z 278.218,A -85,B 0,C 180,E1 -2955.934,E2 -2955.934} C_VEL
LIN {X 0,Y 560.071,Z 378.894,A -85,B 0,C 180,E1 -2957.244,E2 -2957.244} C_VEL
LIN {X 0,Y 559.942,Z 392.183,A -85,B 0,C 180,E1 -2957.564,E2 -2957.564} C_VEL
LIN {X 0,Y 559.778,Z 404.352,A -85,B 0,C 180,E1 -2957.998,E2 -2957.998} C_VEL
LIN {X 0,Y 559.674,Z 415.796,A -85,B 0,C 180,E1 -2958.546,E2 -2958.546} C_VEL
LIN {X 0,Y 559.488,Z 426.889,A -85,B 0,C 180,E1 -2959.23,E2 -2959.23} C_VEL
LIN {X 0,Y 559.309,Z 437.525,A -85,B 0,C 180,E1 -2960.05,E2 -2960.05} C_VEL
LIN {X 0,Y 559.163,Z 447.095,A -85,B 0,C 180,E1 -2960.96,E2 -2960.96} C_VEL
LIN {X 0,Y 559.049,Z 454.952,A -85,B 0,C 180,E1 -2961.868,E2 -2961.868} C_VEL
LIN {X 0,Y 558.942,Z 462.616,A -85,B 0,C 180,E1 -2962.957,E2 -2962.957} C_VEL
LIN {X 0,Y 558.936,Z 469.674,A -85,B 0,C 180,E1 -2964.226,E2 -2964.226} C_VEL
LIN {X 0,Y 558.827,Z 474.368,A -85,B 0,C 180,E1 -2965.31,E2 -2965.31} C_VEL
LIN {X 0,Y 558.837,Z 477.955,A -85,B 0,C 180,E1 -2966.394,E2 -2966.394} C_VEL
LIN {X 0,Y 558.8,Z 479.805,A -85,B 0,C 180,E1 -2967.115,E2 -2967.115} C_VEL
LIN {X 0,Y 558.745,Z 482.182,A -85,B 0,C 180,E1 -2968.557,E2 -2968.557} C_VEL
LIN {X 0,Y 558.74,Z 483,A -85,B 0,C 180,E1 -2969.999,E2 -2969.999} C_VEL
LIN {X 0,Y 558.745,Z 482.186,A -85,B 0,C 180,E1 -2971.44,E2 -2971.44} C_VEL
LIN {X 0,Y 558.8,Z 479.813,A -85,B 0,C 180,E1 -2972.882,E2 -2972.882} C_VEL
LIN {X 0,Y 558.844,Z 476.899,A -85,B 0,C 180,E1 -2973.965,E2 -2973.965} C_VEL
LIN {X 0,Y 558.798,Z 472.953,A -85,B 0,C 180,E1 -2975.05,E2 -2975.05} C_VEL
LIN {X 0,Y 558.922,Z 467.873,A -85,B 0,C 180,E1 -2976.134,E2 -2976.134} C_VEL
LIN {X 0,Y 558.975,Z 461.475,A -85,B 0,C 180,E1 -2977.222,E2 -2977.222} C_VEL
LIN {X 0,Y 559.091,Z 453.487,A -85,B 0,C 180,E1 -2978.311,E2 -2978.311} C_VEL
LIN {X 0,Y 559.185,Z 445.346,A -85,B 0,C 180,E1 -2979.22,E2 -2979.22} C_VEL
LIN {X 0,Y 559.343,Z 435.412,A -85,B 0,C 180,E1 -2980.13,E2 -2980.13} C_VEL
LIN {X 0,Y 559.554,Z 424.382,A -85,B 0,C 180,E1 -2980.938,E2 -2980.938} C_VEL
LIN {X 0,Y 559.704,Z 412.163,A -85,B 0,C 180,E1 -2981.642,E2 -2981.642} C_VEL
LIN {X 0,Y 559.829,Z 399.803,A -85,B 0,C 180,E1 -2982.183,E2 -2982.183} C_VEL
LIN {X 0,Y 559.981,Z 386.394,A -85,B 0,C 180,E1 -2982.594,E2 -2982.594} C_VEL
LIN {X 0,Y 560.068,Z 373.172,A -85,B 0,C 180,E1 -2982.845,E2 -2982.845} C_VEL
LIN {X 0,Y 560.185,Z 276.856,A -85,B 0,C 180,E1 -2984.087,E2 -2984.087} C_VEL
LIN {X 0,Y 559.381,Z 271.344,A -85,B 0,C 180,E1 -2984.203,E2 -2984.203} C_VEL
LIN {X 0,Y 559.488,Z 256.691,A -85,B 0,C 180,E1 -2986.416,E2 -2986.416} C_VEL
LIN {X 0,Y 559.694,Z 240.901,A -85,B 0,C 180,E1 -2988.864,E2 -2988.864} C_VEL
LIN {X 0,Y 559.957,Z 222.463,A -85,B 0,C 180,E1 -2991.754,E2 -2991.754} C_VEL
LIN {X 0,Y 559.183,Z 217.379,A -85,B 0,C 180,E1 -2992.636,E2 -2992.636} C_VEL
LIN {X 0,Y 559.18,Z 217.331,A -85,B 0,C 180,E1 -2996.096,E2 -2996.096} C_VEL
LIN {X 0,Y 559.139,Z 217.331,A -85,B 0,C 180,E1 -2998.529,E2 -2998.529} C_VEL
LIN {X 0,Y 559.147,Z 217.331,A -85,B 0,C 180,E1 -3001.272,E2 -3001.272} C_VEL
LIN {X 0,Y 559.165,Z 217.338,A -85,B 0,C 180,E1 -3003.947,E2 -3003.947} C_VEL
LIN {X 0,Y 559.129,Z 217.332,A -85,B 0,C 180,E1 -3007.108,E2 -3007.108} C_VEL
LIN {X 0,Y 559.158,Z 217.335,A -85,B 0,C 180,E1 -3009.94,E2 -3009.94} C_VEL
LIN {X 0,Y 559.151,Z 217.33,A -85,B 0,C 180,E1 -3012.742,E2 -3012.742} C_VEL
LIN {X 0,Y 559.144,Z 217.331,A -85,B 0,C 180,E1 -3015.76,E2 -3015.76} C_VEL
LIN {X 0,Y 559.157,Z 217.334,A -85,B 0,C 180,E1 -3018.227,E2 -3018.227} C_VEL
LIN {X 0,Y 559.167,Z 217.327,A -85,B 0,C 180,E1 -3021.19,E2 -3021.19} C_VEL
LIN {X 0,Y 559.116,Z 217.333,A -85,B 0,C 180,E1 -3023.786,E2 -3023.786} C_VEL
LIN {X 0,Y 559.156,Z 217.336,A -85,B 0,C 180,E1 -3026.423,E2 -3026.423} C_VEL
LIN {X 0,Y 559.143,Z 217.335,A -85,B 0,C 180,E1 -3028.978,E2 -3028.978} C_VEL
LIN {X 0,Y 559.127,Z 217.331,A -85,B 0,C 180,E1 -3031.623,E2 -3031.623} C_VEL
LIN {X 0,Y 559.151,Z 217.328,A -85,B 0,C 180,E1 -3033.899,E2 -3033.899} C_VEL
LIN {X 0,Y 559.104,Z 217.341,A -85,B 0,C 180,E1 -3037.064,E2 -3037.064} C_VEL
LIN {X 0,Y 559.162,Z 217.33,A -85,B 0,C 180,E1 -3039.393,E2 -3039.393} C_VEL
LIN {X 0,Y 559.116,Z 217.334,A -85,B 0,C 180,E1 -3041.683,E2 -3041.683} C_VEL
LIN {X 0,Y 559.132,Z 217.33,A -85,B 0,C 180,E1 -3043.945,E2 -3043.945} C_VEL
LIN {X 0,Y 559.131,Z 217.337,A -85,B 0,C 180,E1 -3046.921,E2 -3046.921} C_VEL
LIN {X 0,Y 559.17,Z 217.334,A -85,B 0,C 180,E1 -3049.131,E2 -3049.131} C_VEL
LIN {X 0,Y 559.123,Z 217.331,A -85,B 0,C 180,E1 -3052.05,E2 -3052.05} C_VEL
LIN {X 0,Y 559.186,Z 217.324,A -85,B 0,C 180,E1 -3054.227,E2 -3054.227} C_VEL
LIN {X 0,Y 559.21,Z 217.325,A -85,B 0,C 180,E1 -3057.116,E2 -3057.116} C_VEL
LIN {X 0,Y 559.221,Z 217.322,A -85,B 0,C 180,E1 -3059.997,E2 -3059.997} C_VEL
LIN {X 0,Y 559.195,Z 217.324,A -85,B 0,C 180,E1 -3062.879,E2 -3062.879} C_VEL
LIN {X 0,Y 559.188,Z 217.333,A -85,B 0,C 180,E1 -3065.768,E2 -3065.768} C_VEL
LIN {X 0,Y 559.14,Z 217.329,A -85,B 0,C 180,E1 -3068.672,E2 -3068.672} C_VEL
LIN {X 0,Y 559.18,Z 217.331,A -85,B 0,C 180,E1 -3071.598,E2 -3071.598} C_VEL
LIN {X 0,Y 559.158,Z 217.329,A -85,B 0,C 180,E1 -3074.585,E2 -3074.585} C_VEL
LIN {X 0,Y 559.109,Z 217.336,A -85,B 0,C 180,E1 -3077.555,E2 -3077.555} C_VEL
LIN {X 0,Y 559.14,Z 217.336,A -85,B 0,C 180,E1 -3079.835,E2 -3079.835} C_VEL
LIN {X 0,Y 559.116,Z 217.343,A -85,B 0,C 180,E1 -3082.15,E2 -3082.15} C_VEL
LIN {X 0,Y 559.146,Z 217.329,A -85,B 0,C 180,E1 -3085.295,E2 -3085.295} C_VEL
LIN {X 0,Y 559.138,Z 217.337,A -85,B 0,C 180,E1 -3088.379,E2 -3088.379} C_VEL
LIN {X 0,Y 559.109,Z 217.336,A -85,B 0,C 180,E1 -3090.568,E2 -3090.568} C_VEL
LIN {X 0,Y 558.445,Z 217.419,A -85,B 0,C 180,E1 -3091.17,E2 -3091.17} C_VEL
LIN {X 0,Y 555.587,Z 217.779,A -85,B 0,C 180,E1 -3092.146,E2 -3092.146} C_VEL
LIN {X 0,Y 553.178,Z 218.076,A -85,B 0,C 180,E1 -3092.932,E2 -3092.932} C_VEL
LIN {X 0,Y 552.157,Z 218.2,A -85,B 0,C 180,E1 -3093.538,E2 -3093.538} C_VEL
LIN {X 0,Y 552.082,Z 218.21,A -85,B 0,C 180,E1 -3093.744,E2 -3093.744} C_VEL
LIN {X 0,Y 552.084,Z 218.217,A -85,B 0,C 180,E1 -3096.744,E2 -3096.744} C_VEL
LIN {X 0,Y 552.1,Z 218.208,A -85,B 0,C 180,E1 -3099.524,E2 -3099.524} C_VEL
LIN {X 0,Y 552.135,Z 218.205,A -85,B 0,C 180,E1 -3101.439,E2 -3101.439} C_VEL
LIN {X 0,Y 552.058,Z 218.22,A -85,B 0,C 180,E1 -3104.53,E2 -3104.53} C_VEL
LIN {X 0,Y 552.102,Z 218.214,A -85,B 0,C 180,E1 -3107.581,E2 -3107.581} C_VEL
LIN {X 0,Y 552.128,Z 218.252,A -85,B 0,C 180,E1 -3108.068,E2 -3108.068} C_VEL
LIN {X 0,Y 552.654,Z 222.511,A -85,B 0,C 180,E1 -3108.861,E2 -3108.861} C_VEL
LIN {X 0,Y 552.396,Z 239.828,A -85,B 0,C 180,E1 -3111.789,E2 -3111.789} C_VEL
LIN {X 0,Y 552.222,Z 256.699,A -85,B 0,C 180,E1 -3114.632,E2 -3114.632} C_VEL
LIN {X 0,Y 552.403,Z 258.202,A -85,B 0,C 180,E1 -3114.704,E2 -3114.704} C_VEL
LIN {X 0,Y 553.395,Z 265.259,A -85,B 0,C 180,E1 -3114.826,E2 -3114.826} C_VEL
LIN {X 0,Y 553.138,Z 364.3,A -85,B 0,C 180,E1 -3116.135,E2 -3116.135} C_VEL
LIN {X 0,Y 552.978,Z 377.714,A -85,B 0,C 180,E1 -3116.466,E2 -3116.466} C_VEL
LIN {X 0,Y 552.844,Z 390.299,A -85,B 0,C 180,E1 -3116.929,E2 -3116.929} C_VEL
LIN {X 0,Y 552.625,Z 401.893,A -85,B 0,C 180,E1 -3117.506,E2 -3117.506} C_VEL
LIN {X 0,Y 552.421,Z 413.223,A -85,B 0,C 180,E1 -3118.231,E2 -3118.231} C_VEL
LIN {X 0,Y 552.291,Z 423.894,A -85,B 0,C 180,E1 -3119.086,E2 -3119.086} C_VEL
LIN {X 0,Y 552.159,Z 432.51,A -85,B 0,C 180,E1 -3119.932,E2 -3119.932} C_VEL
LIN {X 0,Y 551.988,Z 440.329,A -85,B 0,C 180,E1 -3120.858,E2 -3120.858} C_VEL
LIN {X 0,Y 551.919,Z 447.498,A -85,B 0,C 180,E1 -3121.893,E2 -3121.893} C_VEL
LIN {X 0,Y 551.79,Z 454.007,A -85,B 0,C 180,E1 -3123.061,E2 -3123.061} C_VEL
LIN {X 0,Y 551.745,Z 459.536,A -85,B 0,C 180,E1 -3124.338,E2 -3124.338} C_VEL
LIN {X 0,Y 551.705,Z 463.395,A -85,B 0,C 180,E1 -3125.545,E2 -3125.545} C_VEL
LIN {X 0,Y 551.663,Z 466.019,A -85,B 0,C 180,E1 -3126.74,E2 -3126.74} C_VEL
LIN {X 0,Y 551.632,Z 467.124,A -85,B 0,C 180,E1 -3127.531,E2 -3127.531} C_VEL
LIN {X 0,Y 551.645,Z 467.856,A -85,B 0,C 180,E1 -3128.425,E2 -3128.425} C_VEL
LIN {X 0,Y 551.638,Z 467.994,A -85,B 0,C 180,E1 -3129.102,E2 -3129.102} C_VEL
LIN {X 0,Y 551.676,Z 467.191,A -85,B 0,C 180,E1 -3130.497,E2 -3130.497} C_VEL
LIN {X 0,Y 551.65,Z 465.877,A -85,B 0,C 180,E1 -3131.429,E2 -3131.429} C_VEL
LIN {X 0,Y 551.712,Z 462.644,A -85,B 0,C 180,E1 -3132.805,E2 -3132.805} C_VEL
LIN {X 0,Y 551.752,Z 458.157,A -85,B 0,C 180,E1 -3134.107,E2 -3134.107} C_VEL
LIN {X 0,Y 551.83,Z 452.945,A -85,B 0,C 180,E1 -3135.245,E2 -3135.245} C_VEL
LIN {X 0,Y 551.917,Z 446.364,A -85,B 0,C 180,E1 -3136.376,E2 -3136.376} C_VEL
LIN {X 0,Y 552.002,Z 438.18,A -85,B 0,C 180,E1 -3137.501,E2 -3137.501} C_VEL
LIN {X 0,Y 552.157,Z 429.046,A -85,B 0,C 180,E1 -3138.518,E2 -3138.518} C_VEL
LIN {X 0,Y 552.353,Z 419.629,A -85,B 0,C 180,E1 -3139.37,E2 -3139.37} C_VEL
LIN {X 0,Y 552.53,Z 408.109,A -85,B 0,C 180,E1 -3140.206,E2 -3140.206} C_VEL
LIN {X 0,Y 552.741,Z 396.796,A -85,B 0,C 180,E1 -3140.856,E2 -3140.856} C_VEL
LIN {X 0,Y 552.93,Z 385.274,A -85,B 0,C 180,E1 -3141.366,E2 -3141.366} C_VEL
LIN {X 0,Y 553.031,Z 372.134,A -85,B 0,C 180,E1 -3141.782,E2 -3141.782} C_VEL
LIN {X 0,Y 553.151,Z 359.019,A -85,B 0,C 180,E1 -3142.041,E2 -3142.041} C_VEL
LIN {X 0,Y 553.225,Z 263.059,A -85,B 0,C 180,E1 -3143.298,E2 -3143.298} C_VEL
LIN {X 0,Y 552.253,Z 257.129,A -85,B 0,C 180,E1 -3143.424,E2 -3143.424} C_VEL
LIN {X 0,Y 552.252,Z 252.546,A -85,B 0,C 180,E1 -3144.158,E2 -3144.158} C_VEL
LIN {X 0,Y 552.601,Z 235.547,A -85,B 0,C 180,E1 -3147.085,E2 -3147.085} C_VEL
LIN {X 0,Y 552.742,Z 221.953,A -85,B 0,C 180,E1 -3149.455,E2 -3149.455} C_VEL
LIN {X 0,Y 552.178,Z 218.248,A -85,B 0,C 180,E1 -3150.183,E2 -3150.183} C_VEL
LIN {X 0,Y 552.168,Z 218.205,A -85,B 0,C 180,E1 -3152.919,E2 -3152.919} C_VEL
LIN {X 0,Y 552.161,Z 218.204,A -85,B 0,C 180,E1 -3155.845,E2 -3155.845} C_VEL
LIN {X 0,Y 552.115,Z 218.205,A -85,B 0,C 180,E1 -3158.787,E2 -3158.787} C_VEL
LIN {X 0,Y 552.119,Z 218.212,A -85,B 0,C 180,E1 -3161.752,E2 -3161.752} C_VEL
LIN {X 0,Y 552.085,Z 218.208,A -85,B 0,C 180,E1 -3164.751,E2 -3164.751} C_VEL
LIN {X 0,Y 552.07,Z 218.221,A -85,B 0,C 180,E1 -3167.791,E2 -3167.791} C_VEL
LIN {X 0,Y 552.088,Z 218.215,A -85,B 0,C 180,E1 -3170.104,E2 -3170.104} C_VEL
LIN {X 0,Y 552.051,Z 218.215,A -85,B 0,C 180,E1 -3172.454,E2 -3172.454} C_VEL
LIN {X 0,Y 552.083,Z 218.209,A -85,B 0,C 180,E1 -3175.346,E2 -3175.346} C_VEL
LIN {X 0,Y 552.06,Z 218.215,A -85,B 0,C 180,E1 -3178.56,E2 -3178.56} C_VEL
LIN {X 0,Y 552.077,Z 218.21,A -85,B 0,C 180,E1 -3181.479,E2 -3181.479} C_VEL
LIN {X 0,Y 552.063,Z 218.219,A -85,B 0,C 180,E1 -3184.168,E2 -3184.168} C_VEL
LIN {X 0,Y 552.063,Z 218.216,A -85,B 0,C 180,E1 -3186.751,E2 -3186.751} C_VEL
LIN {X 0,Y 552.095,Z 218.207,A -85,B 0,C 180,E1 -3189.531,E2 -3189.531} C_VEL
LIN {X 0,Y 552.081,Z 218.216,A -85,B 0,C 180,E1 -3192.431,E2 -3192.431} C_VEL
LIN {X 0,Y 552.066,Z 218.211,A -85,B 0,C 180,E1 -3195.566,E2 -3195.566} C_VEL
LIN {X 0,Y 552.051,Z 218.219,A -85,B 0,C 180,E1 -3198.553,E2 -3198.553} C_VEL
LIN {X 0,Y 552.093,Z 218.21,A -85,B 0,C 180,E1 -3201.414,E2 -3201.414} C_VEL
LIN {X 0,Y 552.066,Z 218.211,A -85,B 0,C 180,E1 -3204.16,E2 -3204.16} C_VEL
LIN {X 0,Y 552.087,Z 218.214,A -85,B 0,C 180,E1 -3206.817,E2 -3206.817} C_VEL
LIN {X 0,Y 552.074,Z 218.216,A -85,B 0,C 180,E1 -3209.394,E2 -3209.394} C_VEL
LIN {X 0,Y 552.049,Z 218.214,A -85,B 0,C 180,E1 -3211.903,E2 -3211.903} C_VEL
LIN {X 0,Y 552.067,Z 218.212,A -85,B 0,C 180,E1 -3214.671,E2 -3214.671} C_VEL
LIN {X 0,Y 552.08,Z 218.217,A -85,B 0,C 180,E1 -3217.553,E2 -3217.553} C_VEL
LIN {X 0,Y 552.139,Z 218.202,A -85,B 0,C 180,E1 -3220.379,E2 -3220.379} C_VEL
LIN {X 0,Y 552.101,Z 218.208,A -85,B 0,C 180,E1 -3222.979,E2 -3222.979} C_VEL
LIN {X 0,Y 552.121,Z 218.209,A -85,B 0,C 180,E1 -3226.008,E2 -3226.008} C_VEL
LIN {X 0,Y 552.125,Z 218.204,A -85,B 0,C 180,E1 -3228.996,E2 -3228.996} C_VEL
LIN {X 0,Y 552.112,Z 218.215,A -85,B 0,C 180,E1 -3231.954,E2 -3231.954} C_VEL
LIN {X 0,Y 552.206,Z 218.193,A -85,B 0,C 180,E1 -3234.892,E2 -3234.892} C_VEL
LIN {X 0,Y 552.219,Z 218.197,A -85,B 0,C 180,E1 -3237.815,E2 -3237.815} C_VEL
LIN {X 0,Y 552.24,Z 218.191,A -85,B 0,C 180,E1 -3240.732,E2 -3240.732} C_VEL
LIN {X 0,Y 552.191,Z 218.196,A -85,B 0,C 180,E1 -3242.921,E2 -3242.921} C_VEL
LIN {X 0,Y 552.177,Z 218.2,A -85,B 0,C 180,E1 -3245.847,E2 -3245.847} C_VEL
LIN {X 0,Y 552.135,Z 218.207,A -85,B 0,C 180,E1 -3248.789,E2 -3248.789} C_VEL
LIN {X 0,Y 552.168,Z 218.198,A -85,B 0,C 180,E1 -3251.753,E2 -3251.753} C_VEL
LIN {X 0,Y 552.133,Z 218.211,A -85,B 0,C 180,E1 -3254.751,E2 -3254.751} C_VEL
LIN {X 0,Y 552.101,Z 218.206,A -85,B 0,C 180,E1 -3257.791,E2 -3257.791} C_VEL
LIN {X 0,Y 552.135,Z 218.203,A -85,B 0,C 180,E1 -3260.103,E2 -3260.103} C_VEL
LIN {X 0,Y 552.095,Z 218.211,A -85,B 0,C 180,E1 -3262.453,E2 -3262.453} C_VEL
LIN {X 0,Y 552.095,Z 218.212,A -85,B 0,C 180,E1 -3265.335,E2 -3265.335} C_VEL
LIN {X 0,Y 552.068,Z 218.21,A -85,B 0,C 180,E1 -3268.103,E2 -3268.103} C_VEL
LIN {X 0,Y 552.104,Z 218.208,A -85,B 0,C 180,E1 -3270.611,E2 -3270.611} C_VEL
LIN {X 0,Y 552.116,Z 218.214,A -85,B 0,C 180,E1 -3273.188,E2 -3273.188} C_VEL
LIN {X 0,Y 552.083,Z 218.211,A -85,B 0,C 180,E1 -3275.846,E2 -3275.846} C_VEL
LIN {X 0,Y 552.125,Z 218.204,A -85,B 0,C 180,E1 -3278.59,E2 -3278.59} C_VEL
LIN {X 0,Y 552.089,Z 218.218,A -85,B 0,C 180,E1 -3281.451,E2 -3281.451} C_VEL
LIN {X 0,Y 552.087,Z 218.208,A -85,B 0,C 180,E1 -3284.53,E2 -3284.53} C_VEL
LIN {X 0,Y 552.099,Z 218.215,A -85,B 0,C 180,E1 -3287.59,E2 -3287.59} C_VEL
LIN {X 0,Y 552.138,Z 218.203,A -85,B 0,C 180,E1 -3290.473,E2 -3290.473} C_VEL
LIN {X 0,Y 552.109,Z 218.207,A -85,B 0,C 180,E1 -3293.318,E2 -3293.318} C_VEL
LIN {X 0,Y 552.135,Z 218.212,A -85,B 0,C 180,E1 -3295.939,E2 -3295.939} C_VEL
LIN {X 0,Y 552.132,Z 218.205,A -85,B 0,C 180,E1 -3298.54,E2 -3298.54} C_VEL
LIN {X 0,Y 552.113,Z 218.207,A -85,B 0,C 180,E1 -3301.442,E2 -3301.442} C_VEL
LIN {X 0,Y 552.116,Z 218.208,A -85,B 0,C 180,E1 -3303.542,E2 -3303.542} C_VEL
LIN {X 0,Y 552.104,Z 218.215,A -85,B 0,C 180,E1 -3306.757,E2 -3306.757} C_VEL
LIN {X 0,Y 552.133,Z 218.327,A -85,B 0,C 180,E1 -3307.204,E2 -3307.204} C_VEL
LIN {X 0,Y 552.999,Z 223.332,A -85,B 0,C 180,E1 -3308.088,E2 -3308.088} C_VEL
LIN {X 0,Y 552.732,Z 239.644,A -85,B 0,C 180,E1 -3310.694,E2 -3310.694} C_VEL
LIN {X 0,Y 552.517,Z 255.399,A -85,B 0,C 180,E1 -3313.178,E2 -3313.178} C_VEL
LIN {X 0,Y 552.363,Z 271.25,A -85,B 0,C 180,E1 -3315.612,E2 -3315.612} C_VEL
LIN {X 0,Y 553.436,Z 278.917,A -85,B 0,C 180,E1 -3315.766,E2 -3315.766} C_VEL
LIN {X 0,Y 553.159,Z 378.856,A -85,B 0,C 180,E1 -3317.082,E2 -3317.082} C_VEL
LIN {X 0,Y 553.021,Z 392.16,A -85,B 0,C 180,E1 -3317.406,E2 -3317.406} C_VEL
LIN {X 0,Y 552.826,Z 404.335,A -85,B 0,C 180,E1 -3317.844,E2 -3317.844} C_VEL
LIN {X 0,Y 552.696,Z 416.645,A -85,B 0,C 180,E1 -3318.448,E2 -3318.448} C_VEL
LIN {X 0,Y 552.49,Z 428.178,A -85,B 0,C 180,E1 -3319.185,E2 -3319.185} C_VEL
LIN {X 0,Y 552.294,Z 438.592,A -85,B 0,C 180,E1 -3320.015,E2 -3320.015} C_VEL
LIN {X 0,Y 552.127,Z 447.103,A -85,B 0,C 180,E1 -3320.844,E2 -3320.844} C_VEL
LIN {X 0,Y 552.011,Z 454.952,A -85,B 0,C 180,E1 -3321.764,E2 -3321.764} C_VEL
LIN {X 0,Y 551.89,Z 462.615,A -85,B 0,C 180,E1 -3322.867,E2 -3322.867} C_VEL
LIN {X 0,Y 551.869,Z 469.674,A -85,B 0,C 180,E1 -3324.152,E2 -3324.152} C_VEL
LIN {X 0,Y 551.725,Z 474.369,A -85,B 0,C 180,E1 -3325.249,E2 -3325.249} C_VEL
LIN {X 0,Y 551.751,Z 477.955,A -85,B 0,C 180,E1 -3326.347,E2 -3326.347} C_VEL
LIN {X 0,Y 551.724,Z 479.804,A -85,B 0,C 180,E1 -3327.078,E2 -3327.078} C_VEL
LIN {X 0,Y 551.645,Z 482.181,A -85,B 0,C 180,E1 -3328.539,E2 -3328.539} C_VEL
LIN {X 0,Y 551.64,Z 483,A -85,B 0,C 180,E1 -3329.999,E2 -3329.999} C_VEL
LIN {X 0,Y 551.645,Z 482.185,A -85,B 0,C 180,E1 -3331.459,E2 -3331.459} C_VEL
LIN {X 0,Y 551.724,Z 479.813,A -85,B 0,C 180,E1 -3332.919,E2 -3332.919} C_VEL
LIN {X 0,Y 551.764,Z 476.899,A -85,B 0,C 180,E1 -3334.016,E2 -3334.016} C_VEL
LIN {X 0,Y 551.724,Z 472.953,A -85,B 0,C 180,E1 -3335.115,E2 -3335.115} C_VEL
LIN {X 0,Y 551.816,Z 467.133,A -85,B 0,C 180,E1 -3336.351,E2 -3336.351} C_VEL
LIN {X 0,Y 551.927,Z 460.243,A -85,B 0,C 180,E1 -3337.498,E2 -3337.498} C_VEL
LIN {X 0,Y 552.064,Z 452.002,A -85,B 0,C 180,E1 -3338.601,E2 -3338.601} C_VEL
LIN {X 0,Y 552.222,Z 443.552,A -85,B 0,C 180,E1 -3339.522,E2 -3339.522} C_VEL
LIN {X 0,Y 552.4,Z 433.107,A -85,B 0,C 180,E1 -3340.444,E2 -3340.444} C_VEL
LIN {X 0,Y 552.616,Z 422.146,A -85,B 0,C 180,E1 -3341.222,E2 -3341.222} C_VEL
LIN {X 0,Y 552.783,Z 411.427,A -85,B 0,C 180,E1 -3341.829,E2 -3341.829} C_VEL
LIN {X 0,Y 552.885,Z 399.785,A -85,B 0,C 180,E1 -3342.339,E2 -3342.339} C_VEL
LIN {X 0,Y 553.073,Z 386.362,A -85,B 0,C 180,E1 -3342.754,E2 -3342.754} C_VEL
LIN {X 0,Y 553.17,Z 373.12,A -85,B 0,C 180,E1 -3343.008,E2 -3343.008} C_VEL
LIN {X 0,Y 553.323,Z 277.784,A -85,B 0,C 180,E1 -3344.252,E2 -3344.252} C_VEL
LIN {X 0,Y 552.385,Z 271.274,A -85,B 0,C 180,E1 -3344.386,E2 -3344.386} C_VEL
LIN {X 0,Y 552.475,Z 256.583,A -85,B 0,C 180,E1 -3346.631,E2 -3346.631} C_VEL
LIN {X 0,Y 552.7,Z 241.994,A -85,B 0,C 180,E1 -3348.919,E2 -3348.919} C_VEL
LIN {X 0,Y 552.98,Z 224.926,A -85,B 0,C 180,E1 -3351.626,E2 -3351.626} C_VEL
LIN {X 0,Y 552.445,Z 220.024,A -85,B 0,C 180,E1 -3352.434,E2 -3352.434} C_VEL
LIN {X 0,Y 552.136,Z 218.243,A -85,B 0,C 180,E1 -3352.793,E2 -3352.793} C_VEL
LIN {X 0,Y 552.12,Z 218.215,A -85,B 0,C 180,E1 -3355.643,E2 -3355.643} C_VEL
LIN {X 0,Y 552.107,Z 218.212,A -85,B 0,C 180,E1 -3358.097,E2 -3358.097} C_VEL
LIN {X 0,Y 552.101,Z 218.208,A -85,B 0,C 180,E1 -3360.608,E2 -3360.608} C_VEL
LIN {X 0,Y 552.115,Z 218.206,A -85,B 0,C 180,E1 -3363.184,E2 -3363.184} C_VEL
LIN {X 0,Y 552.074,Z 218.217,A -85,B 0,C 180,E1 -3365.843,E2 -3365.843} C_VEL
LIN {X 0,Y 552.113,Z 218.208,A -85,B 0,C 180,E1 -3368.587,E2 -3368.587} C_VEL
LIN {X 0,Y 552.118,Z 218.205,A -85,B 0,C 180,E1 -3371.444,E2 -3371.444} C_VEL
LIN {X 0,Y 552.086,Z 218.214,A -85,B 0,C 180,E1 -3374.529,E2 -3374.529} C_VEL
LIN {X 0,Y 552.107,Z 218.204,A -85,B 0,C 180,E1 -3377.585,E2 -3377.585} C_VEL
LIN {X 0,Y 552.124,Z 218.213,A -85,B 0,C 180,E1 -3380.471,E2 -3380.471} C_VEL
LIN {X 0,Y 552.094,Z 218.207,A -85,B 0,C 180,E1 -3383.316,E2 -3383.316} C_VEL
LIN {X 0,Y 552.12,Z 218.206,A -85,B 0,C 180,E1 -3385.937,E2 -3385.937} C_VEL
LIN {X 0,Y 552.115,Z 218.213,A -85,B 0,C 180,E1 -3388.538,E2 -3388.538} C_VEL
LIN {X 0,Y 552.089,Z 218.209,A -85,B 0,C 180,E1 -3391.442,E2 -3391.442} C_VEL
LIN {X 0,Y 552.076,Z 218.213,A -85,B 0,C 180,E1 -3394.351,E2 -3394.351} C_VEL
LIN {X 0,Y 552.081,Z 218.217,A -85,B 0,C 180,E1 -3396.755,E2 -3396.755} C_VEL
LIN {X 0,Y 552.107,Z 218.213,A -85,B 0,C 180,E1 -3399.117,E2 -3399.117} C_VEL
LIN {X 0,Y 552.076,Z 218.213,A -85,B 0,C 180,E1 -3401.44,E2 -3401.44} C_VEL
LIN {X 0,Y 552.081,Z 218.209,A -85,B 0,C 180,E1 -3403.734,E2 -3403.734} C_VEL
LIN {X 0,Y 552.096,Z 218.208,A -85,B 0,C 180,E1 -3406.001,E2 -3406.001} C_VEL
LIN {X 0,Y 552.141,Z 218.207,A -85,B 0,C 180,E1 -3408.991,E2 -3408.991} C_VEL
LIN {X 0,Y 552.093,Z 218.207,A -85,B 0,C 180,E1 -3411.948,E2 -3411.948} C_VEL
LIN {X 0,Y 552.159,Z 218.2,A -85,B 0,C 180,E1 -3414.153,E2 -3414.153} C_VEL
LIN {X 0,Y 552.174,Z 218.201,A -85,B 0,C 180,E1 -3417.079,E2 -3417.079} C_VEL
LIN {X 0,Y 552.192,Z 218.198,A -85,B 0,C 180,E1 -3419.997,E2 -3419.997} C_VEL
LIN {X 0,Y 552.164,Z 218.2,A -85,B 0,C 180,E1 -3422.915,E2 -3422.915} C_VEL
LIN {X 0,Y 552.157,Z 218.207,A -85,B 0,C 180,E1 -3425.841,E2 -3425.841} C_VEL
LIN {X 0,Y 552.113,Z 218.205,A -85,B 0,C 180,E1 -3428.783,E2 -3428.783} C_VEL
LIN {X 0,Y 552.135,Z 218.211,A -85,B 0,C 180,E1 -3431.748,E2 -3431.748} C_VEL
LIN {X 0,Y 552.105,Z 218.207,A -85,B 0,C 180,E1 -3434.746,E2 -3434.746} C_VEL
LIN {X 0,Y 552.067,Z 218.217,A -85,B 0,C 180,E1 -3437.786,E2 -3437.786} C_VEL
LIN {X 0,Y 552.101,Z 218.216,A -85,B 0,C 180,E1 -3440.099,E2 -3440.099} C_VEL
LIN {X 0,Y 552.067,Z 218.216,A -85,B 0,C 180,E1 -3442.448,E2 -3442.448} C_VEL
LIN {X 0,Y 552.108,Z 218.205,A -85,B 0,C 180,E1 -3445.344,E2 -3445.344} C_VEL
LIN {X 0,Y 552.08,Z 218.216,A -85,B 0,C 180,E1 -3448.096,E2 -3448.096} C_VEL
LIN {X 0,Y 552.072,Z 218.217,A -85,B 0,C 180,E1 -3450.607,E2 -3450.607} C_VEL
LIN {X 0,Y 552.091,Z 218.209,A -85,B 0,C 180,E1 -3453.183,E2 -3453.183} C_VEL
LIN {X 0,Y 552.082,Z 218.21,A -85,B 0,C 180,E1 -3453.744,E2 -3453.744} C_VEL
LIN {X 0,Y 551.445,Z 218.297,A -85,B 0,C 180,E1 -3454.352,E2 -3454.352} C_VEL
LIN {X 0,Y 548.631,Z 218.65,A -85,B 0,C 180,E1 -3455.341,E2 -3455.341} C_VEL
LIN {X 0,Y 546.216,Z 218.951,A -85,B 0,C 180,E1 -3456.137,E2 -3456.137} C_VEL
LIN {X 0,Y 545.145,Z 219.081,A -85,B 0,C 180,E1 -3456.751,E2 -3456.751} C_VEL
LIN {X 0,Y 545.041,Z 219.091,A -85,B 0,C 180,E1 -3456.959,E2 -3456.959} C_VEL
LIN {X 0,Y 545.059,Z 219.088,A -85,B 0,C 180,E1 -3460.138,E2 -3460.138} C_VEL
LIN {X 0,Y 545.031,Z 219.097,A -85,B 0,C 180,E1 -3462.695,E2 -3462.695} C_VEL
LIN {X 0,Y 545.024,Z 219.096,A -85,B 0,C 180,E1 -3465.165,E2 -3465.165} C_VEL
LIN {X 0,Y 545.121,Z 219.141,A -85,B 0,C 180,E1 -3467.971,E2 -3467.971} C_VEL
LIN {X 0,Y 545.663,Z 224.409,A -85,B 0,C 180,E1 -3468.941,E2 -3468.941} C_VEL
LIN {X 0,Y 545.373,Z 241.239,A -85,B 0,C 180,E1 -3471.813,E2 -3471.813} C_VEL
LIN {X 0,Y 545.231,Z 256.979,A -85,B 0,C 180,E1 -3474.463,E2 -3474.463} C_VEL
LIN {X 0,Y 545.924,Z 261.319,A -85,B 0,C 180,E1 -3474.573,E2 -3474.573} C_VEL
LIN {X 0,Y 546.514,Z 266.403,A -85,B 0,C 180,E1 -3474.657,E2 -3474.657} C_VEL
LIN {X 0,Y 546.225,Z 364.263,A -85,B 0,C 180,E1 -3475.967,E2 -3475.967} C_VEL
LIN {X 0,Y 546.061,Z 377.727,A -85,B 0,C 180,E1 -3476.303,E2 -3476.303} C_VEL
LIN {X 0,Y 545.914,Z 390.051,A -85,B 0,C 180,E1 -3476.759,E2 -3476.759} C_VEL
LIN {X 0,Y 545.674,Z 402.083,A -85,B 0,C 180,E1 -3477.364,E2 -3477.364} C_VEL
LIN {X 0,Y 545.432,Z 413.576,A -85,B 0,C 180,E1 -3478.111,E2 -3478.111} C_VEL
LIN {X 0,Y 545.283,Z 424.082,A -85,B 0,C 180,E1 -3478.967,E2 -3478.967} C_VEL
LIN {X 0,Y 545.125,Z 432.585,A -85,B 0,C 180,E1 -3479.816,E2 -3479.816} C_VEL
LIN {X 0,Y 544.922,Z 440.933,A -85,B 0,C 180,E1 -3480.829,E2 -3480.829} C_VEL
LIN {X 0,Y 544.836,Z 448.204,A -85,B 0,C 180,E1 -3481.914,E2 -3481.914} C_VEL
LIN {X 0,Y 544.701,Z 454.856,A -85,B 0,C 180,E1 -3483.156,E2 -3483.156} C_VEL
LIN {X 0,Y 544.665,Z 459.678,A -85,B 0,C 180,E1 -3484.314,E2 -3484.314} C_VEL
LIN {X 0,Y 544.611,Z 463.673,A -85,B 0,C 180,E1 -3485.611,E2 -3485.611} C_VEL
LIN {X 0,Y 544.591,Z 465.469,A -85,B 0,C 180,E1 -3486.42,E2 -3486.42} C_VEL
LIN {X 0,Y 544.533,Z 466.794,A -85,B 0,C 180,E1 -3487.221,E2 -3487.221} C_VEL
LIN {X 0,Y 544.545,Z 467.785,A -85,B 0,C 180,E1 -3488.304,E2 -3488.304} C_VEL
LIN {X 0,Y 544.552,Z 467.883,A -85,B 0,C 180,E1 -3489.608,E2 -3489.608} C_VEL
LIN {X 0,Y 544.583,Z 467.32,A -85,B 0,C 180,E1 -3490.396,E2 -3490.396} C_VEL
LIN {X 0,Y 544.551,Z 466.323,A -85,B 0,C 180,E1 -3491.178,E2 -3491.178} C_VEL
LIN {X 0,Y 544.563,Z 464.903,A -85,B 0,C 180,E1 -3491.958,E2 -3491.958} C_VEL
LIN {X 0,Y 544.635,Z 461.87,A -85,B 0,C 180,E1 -3493.123,E2 -3493.123} C_VEL
LIN {X 0,Y 544.67,Z 457.743,A -85,B 0,C 180,E1 -3494.279,E2 -3494.279} C_VEL
LIN {X 0,Y 544.755,Z 451.591,A -85,B 0,C 180,E1 -3495.581,E2 -3495.581} C_VEL
LIN {X 0,Y 544.853,Z 444.45,A -85,B 0,C 180,E1 -3496.766,E2 -3496.766} C_VEL
LIN {X 0,Y 545,Z 437.382,A -85,B 0,C 180,E1 -3497.716,E2 -3497.716} C_VEL
LIN {X 0,Y 545.154,Z 428.278,A -85,B 0,C 180,E1 -3498.724,E2 -3498.724} C_VEL
LIN {X 0,Y 545.354,Z 418.402,A -85,B 0,C 180,E1 -3499.607,E2 -3499.607} C_VEL
LIN {X 0,Y 545.6,Z 406.594,A -85,B 0,C 180,E1 -3500.455,E2 -3500.455} C_VEL
LIN {X 0,Y 545.809,Z 394.778,A -85,B 0,C 180,E1 -3501.113,E2 -3501.113} C_VEL
LIN {X 0,Y 546.02,Z 382.475,A -85,B 0,C 180,E1 -3501.629,E2 -3501.629} C_VEL
LIN {X 0,Y 546.181,Z 369.383,A -85,B 0,C 180,E1 -3502.016,E2 -3502.016} C_VEL
LIN {X 0,Y 546.278,Z 355.015,A -85,B 0,C 180,E1 -3502.263,E2 -3502.263} C_VEL
LIN {X 0,Y 546.362,Z 264.012,A -85,B 0,C 180,E1 -3503.469,E2 -3503.469} C_VEL
LIN {X 0,Y 545.232,Z 257.143,A -85,B 0,C 180,E1 -3503.618,E2 -3503.618} C_VEL
LIN {X 0,Y 545.475,Z 241.411,A -85,B 0,C 180,E1 -3506.308,E2 -3506.308} C_VEL
LIN {X 0,Y 545.833,Z 224.581,A -85,B 0,C 180,E1 -3509.263,E2 -3509.263} C_VEL
LIN {X 0,Y 545.152,Z 219.148,A -85,B 0,C 180,E1 -3510.301,E2 -3510.301} C_VEL
LIN {X 0,Y 545.135,Z 219.082,A -85,B 0,C 180,E1 -3512.957,E2 -3512.957} C_VEL
LIN {X 0,Y 545.131,Z 219.079,A -85,B 0,C 180,E1 -3515.921,E2 -3515.921} C_VEL
LIN {X 0,Y 545.074,Z 219.083,A -85,B 0,C 180,E1 -3518.902,E2 -3518.902} C_VEL
LIN {X 0,Y 545.091,Z 219.085,A -85,B 0,C 180,E1 -3521.906,E2 -3521.906} C_VEL
LIN {X 0,Y 545.038,Z 219.087,A -85,B 0,C 180,E1 -3524.946,E2 -3524.946} C_VEL
LIN {X 0,Y 545.038,Z 219.093,A -85,B 0,C 180,E1 -3528.028,E2 -3528.028} C_VEL
LIN {X 0,Y 545.053,Z 219.087,A -85,B 0,C 180,E1 -3530.375,E2 -3530.375} C_VEL
LIN {X 0,Y 545.041,Z 219.089,A -85,B 0,C 180,E1 -3533.562,E2 -3533.562} C_VEL
LIN {X 0,Y 545.018,Z 219.098,A -85,B 0,C 180,E1 -3536.005,E2 -3536.005} C_VEL
LIN {X 0,Y 545.032,Z 219.089,A -85,B 0,C 180,E1 -3538.747,E2 -3538.747} C_VEL
LIN {X 0,Y 545.023,Z 219.09,A -85,B 0,C 180,E1 -3541.682,E2 -3541.682} C_VEL
LIN {X 0,Y 545.013,Z 219.096,A -85,B 0,C 180,E1 -3544.569,E2 -3544.569} C_VEL
LIN {X 0,Y 544.993,Z 219.092,A -85,B 0,C 180,E1 -3547.309,E2 -3547.309} C_VEL
LIN {X 0,Y 545.027,Z 219.092,A -85,B 0,C 180,E1 -3550.147,E2 -3550.147} C_VEL
LIN {X 0,Y 544.996,Z 219.094,A -85,B 0,C 180,E1 -3553.116,E2 -3553.116} C_VEL
LIN {X 0,Y 545.025,Z 219.091,A -85,B 0,C 180,E1 -3556.23,E2 -3556.23} C_VEL
LIN {X 0,Y 545.006,Z 219.1,A -85,B 0,C 180,E1 -3558.884,E2 -3558.884} C_VEL
LIN {X 0,Y 545.028,Z 219.088,A -85,B 0,C 180,E1 -3561.766,E2 -3561.766} C_VEL
LIN {X 0,Y 545.017,Z 219.092,A -85,B 0,C 180,E1 -3564.535,E2 -3564.535} C_VEL
LIN {X 0,Y 545.045,Z 219.094,A -85,B 0,C 180,E1 -3567.215,E2 -3567.215} C_VEL
LIN {X 0,Y 545.048,Z 219.086,A -85,B 0,C 180,E1 -3569.814,E2 -3569.814} C_VEL
LIN {X 0,Y 545.014,Z 219.093,A -85,B 0,C 180,E1 -3572.845,E2 -3572.845} C_VEL
LIN {X 0,Y 545.006,Z 219.096,A -85,B 0,C 180,E1 -3575.633,E2 -3575.633} C_VEL
LIN {X 0,Y 545.058,Z 219.084,A -85,B 0,C 180,E1 -3578.184,E2 -3578.184} C_VEL
LIN {X 0,Y 545.11,Z 219.077,A -85,B 0,C 180,E1 -3580.418,E2 -3580.418} C_VEL
LIN {X 0,Y 545.032,Z 219.096,A -85,B 0,C 180,E1 -3583.524,E2 -3583.524} C_VEL
LIN {X 0,Y 545.078,Z 219.09,A -85,B 0,C 180,E1 -3585.823,E2 -3585.823} C_VEL
LIN {X 0,Y 545.071,Z 219.082,A -85,B 0,C 180,E1 -3588.852,E2 -3588.852} C_VEL
LIN {X 0,Y 545.07,Z 219.092,A -85,B 0,C 180,E1 -3591.849,E2 -3591.849} C_VEL
LIN {X 0,Y 545.165,Z 219.071,A -85,B 0,C 180,E1 -3594.826,E2 -3594.826} C_VEL
LIN {X 0,Y 545.191,Z 219.073,A -85,B 0,C 180,E1 -3597.787,E2 -3597.787} C_VEL
LIN {X 0,Y 545.211,Z 219.067,A -85,B 0,C 180,E1 -3600.741,E2 -3600.741} C_VEL
LIN {X 0,Y 545.157,Z 219.072,A -85,B 0,C 180,E1 -3602.959,E2 -3602.959} C_VEL
LIN {X 0,Y 545.131,Z 219.078,A -85,B 0,C 180,E1 -3605.923,E2 -3605.923} C_VEL
LIN {X 0,Y 545.078,Z 219.084,A -85,B 0,C 180,E1 -3608.903,E2 -3608.903} C_VEL
LIN {X 0,Y 545.111,Z 219.079,A -85,B 0,C 180,E1 -3611.907,E2 -3611.907} C_VEL
LIN {X 0,Y 545.09,Z 219.085,A -85,B 0,C 180,E1 -3614.946,E2 -3614.946} C_VEL
LIN {X 0,Y 545.067,Z 219.083,A -85,B 0,C 180,E1 -3618.028,E2 -3618.028} C_VEL
LIN {X 0,Y 545.101,Z 219.082,A -85,B 0,C 180,E1 -3620.374,E2 -3620.374} C_VEL
LIN {X 0,Y 545.082,Z 219.082,A -85,B 0,C 180,E1 -3623.561,E2 -3623.561} C_VEL
LIN {X 0,Y 545.068,Z 219.089,A -85,B 0,C 180,E1 -3626.828,E2 -3626.828} C_VEL
LIN {X 0,Y 545.038,Z 219.093,A -85,B 0,C 180,E1 -3629.342,E2 -3629.342} C_VEL
LIN {X 0,Y 545.058,Z 219.085,A -85,B 0,C 180,E1 -3631.917,E2 -3631.917} C_VEL
LIN {X 0,Y 545.059,Z 219.084,A -85,B 0,C 180,E1 -3634.567,E2 -3634.567} C_VEL
LIN {X 0,Y 545.043,Z 219.095,A -85,B 0,C 180,E1 -3637.305,E2 -3637.305} C_VEL
LIN {X 0,Y 545.071,Z 219.083,A -85,B 0,C 180,E1 -3640.144,E2 -3640.144} C_VEL
LIN {X 0,Y 545.03,Z 219.09,A -85,B 0,C 180,E1 -3643.113,E2 -3643.113} C_VEL
LIN {X 0,Y 545.04,Z 219.088,A -85,B 0,C 180,E1 -3646.229,E2 -3646.229} C_VEL
LIN {X 0,Y 545.04,Z 219.086,A -85,B 0,C 180,E1 -3648.881,E2 -3648.881} C_VEL
LIN {X 0,Y 545.06,Z 219.093,A -85,B 0,C 180,E1 -3651.762,E2 -3651.762} C_VEL
LIN {X 0,Y 545.036,Z 219.088,A -85,B 0,C 180,E1 -3654.531,E2 -3654.531} C_VEL
LIN {X 0,Y 545.077,Z 219.082,A -85,B 0,C 180,E1 -3657.211,E2 -3657.211} C_VEL
LIN {X 0,Y 545.073,Z 219.087,A -85,B 0,C 180,E1 -3659.81,E2 -3659.81} C_VEL
LIN {X 0,Y 545.067,Z 219.092,A -85,B 0,C 180,E1 -3662.342,E2 -3662.342} C_VEL
LIN {X 0,Y 545.053,Z 219.09,A -85,B 0,C 180,E1 -3664.816,E2 -3664.816} C_VEL
LIN {X 0,Y 545.091,Z 219.185,A -85,B 0,C 180,E1 -3667.043,E2 -3667.043} C_VEL
LIN {X 0,Y 546.047,Z 225.005,A -85,B 0,C 180,E1 -3668.083,E2 -3668.083} C_VEL
LIN {X 0,Y 545.756,Z 241.974,A -85,B 0,C 180,E1 -3670.829,E2 -3670.829} C_VEL
LIN {X 0,Y 545.479,Z 257.727,A -85,B 0,C 180,E1 -3673.34,E2 -3673.34} C_VEL
LIN {X 0,Y 545.347,Z 271.122,A -85,B 0,C 180,E1 -3675.421,E2 -3675.421} C_VEL
LIN {X 0,Y 546.458,Z 278.253,A -85,B 0,C 180,E1 -3675.573,E2 -3675.573} C_VEL
LIN {X 0,Y 546.234,Z 378.693,A -85,B 0,C 180,E1 -3676.916,E2 -3676.916} C_VEL
LIN {X 0,Y 546.105,Z 392.02,A -85,B 0,C 180,E1 -3677.244,E2 -3677.244} C_VEL
LIN {X 0,Y 545.874,Z 404.205,A -85,B 0,C 180,E1 -3677.687,E2 -3677.687} C_VEL
LIN {X 0,Y 545.713,Z 416.536,A -85,B 0,C 180,E1 -3678.298,E2 -3678.298} C_VEL
LIN {X 0,Y 545.493,Z 428.092,A -85,B 0,C 180,E1 -3679.044,E2 -3679.044} C_VEL
LIN {X 0,Y 545.251,Z 438.529,A -85,B 0,C 180,E1 -3679.884,E2 -3679.884} C_VEL
LIN {X 0,Y 545.087,Z 447.059,A -85,B 0,C 180,E1 -3680.724,E2 -3680.724} C_VEL
LIN {X 0,Y 544.974,Z 454.929,A -85,B 0,C 180,E1 -3681.657,E2 -3681.657} C_VEL
LIN {X 0,Y 544.826,Z 462.611,A -85,B 0,C 180,E1 -3682.774,E2 -3682.774} C_VEL
LIN {X 0,Y 544.779,Z 469.674,A -85,B 0,C 180,E1 -3684.075,E2 -3684.075} C_VEL
LIN {X 0,Y 544.629,Z 474.369,A -85,B 0,C 180,E1 -3685.187,E2 -3685.187} C_VEL
LIN {X 0,Y 544.67,Z 477.954,A -85,B 0,C 180,E1 -3686.3,E2 -3686.3} C_VEL
LIN {X 0,Y 544.651,Z 479.804,A -85,B 0,C 180,E1 -3687.04,E2 -3687.04} C_VEL
LIN {X 0,Y 544.546,Z 482.18,A -85,B 0,C 180,E1 -3688.52,E2 -3688.52} C_VEL
LIN {X 0,Y 544.541,Z 483,A -85,B 0,C 180,E1 -3689.999,E2 -3689.999} C_VEL
LIN {X 0,Y 544.546,Z 482.184,A -85,B 0,C 180,E1 -3691.478,E2 -3691.478} C_VEL
LIN {X 0,Y 544.651,Z 479.812,A -85,B 0,C 180,E1 -3692.957,E2 -3692.957} C_VEL
LIN {X 0,Y 544.684,Z 476.899,A -85,B 0,C 180,E1 -3694.068,E2 -3694.068} C_VEL
LIN {X 0,Y 544.654,Z 472.952,A -85,B 0,C 180,E1 -3695.181,E2 -3695.181} C_VEL
LIN {X 0,Y 544.731,Z 467.654,A -85,B 0,C 180,E1 -3696.338,E2 -3696.338} C_VEL
LIN {X 0,Y 544.837,Z 461.467,A -85,B 0,C 180,E1 -3697.41,E2 -3697.41} C_VEL
LIN {X 0,Y 544.995,Z 453.459,A -85,B 0,C 180,E1 -3698.527,E2 -3698.527} C_VEL
LIN {X 0,Y 545.153,Z 445.296,A -85,B 0,C 180,E1 -3699.459,E2 -3699.459} C_VEL
LIN {X 0,Y 545.351,Z 435.338,A -85,B 0,C 180,E1 -3700.393,E2 -3700.393} C_VEL
LIN {X 0,Y 545.584,Z 424.458,A -85,B 0,C 180,E1 -3701.21,E2 -3701.21} C_VEL
LIN {X 0,Y 545.769,Z 413.071,A -85,B 0,C 180,E1 -3701.889,E2 -3701.889} C_VEL
LIN {X 0,Y 545.919,Z 400.852,A -85,B 0,C 180,E1 -3702.451,E2 -3702.451} C_VEL
LIN {X 0,Y 546.119,Z 388.034,A -85,B 0,C 180,E1 -3702.872,E2 -3702.872} C_VEL
LIN {X 0,Y 546.244,Z 374.439,A -85,B 0,C 180,E1 -3703.153,E2 -3703.153} C_VEL
LIN {X 0,Y 546.421,Z 278.371,A -85,B 0,C 180,E1 -3704.426,E2 -3704.426} C_VEL
LIN {X 0,Y 545.362,Z 271.149,A -85,B 0,C 180,E1 -3704.576,E2 -3704.576} C_VEL
LIN {X 0,Y 545.627,Z 250.876,A -85,B 0,C 180,E1 -3707.735,E2 -3707.735} C_VEL
LIN {X 0,Y 545.972,Z 229.68,A -85,B 0,C 180,E1 -3711.125,E2 -3711.125} C_VEL
LIN {X 0,Y 545.967,Z 223.96,A -85,B 0,C 180,E1 -3712.053,E2 -3712.053} C_VEL
LIN {X 0,Y 545.08,Z 219.196,A -85,B 0,C 180,E1 -3712.905,E2 -3712.905} C_VEL
LIN {X 0,Y 545.075,Z 219.091,A -85,B 0,C 180,E1 -3715.999,E2 -3715.999} C_VEL
LIN {X 0,Y 545.074,Z 219.083,A -85,B 0,C 180,E1 -3718.743,E2 -3718.743} C_VEL
LIN {X 0,Y 545.059,Z 219.091,A -85,B 0,C 180,E1 -3721.677,E2 -3721.677} C_VEL
LIN {X 0,Y 545.06,Z 219.085,A -85,B 0,C 180,E1 -3724.563,E2 -3724.563} C_VEL
LIN {X 0,Y 545.03,Z 219.089,A -85,B 0,C 180,E1 -3727.303,E2 -3727.303} C_VEL
LIN {X 0,Y 545.063,Z 219.094,A -85,B 0,C 180,E1 -3730.141,E2 -3730.141} C_VEL
LIN {X 0,Y 545.046,Z 219.088,A -85,B 0,C 180,E1 -3732.693,E2 -3732.693} C_VEL
LIN {X 0,Y 545.03,Z 219.087,A -85,B 0,C 180,E1 -3735.168,E2 -3735.168} C_VEL
LIN {X 0,Y 545.06,Z 219.085,A -85,B 0,C 180,E1 -3737.893,E2 -3737.893} C_VEL
LIN {X 0,Y 545.074,Z 219.086,A -85,B 0,C 180,E1 -3740.816,E2 -3740.816} C_VEL
LIN {X 0,Y 545.03,Z 219.087,A -85,B 0,C 180,E1 -3743.617,E2 -3743.617} C_VEL
LIN {X 0,Y 545.059,Z 219.09,A -85,B 0,C 180,E1 -3746.326,E2 -3746.326} C_VEL
LIN {X 0,Y 545.057,Z 219.09,A -85,B 0,C 180,E1 -3748.95,E2 -3748.95} C_VEL
LIN {X 0,Y 545.067,Z 219.083,A -85,B 0,C 180,E1 -3751.504,E2 -3751.504} C_VEL
LIN {X 0,Y 545.03,Z 219.093,A -85,B 0,C 180,E1 -3754.502,E2 -3754.502} C_VEL
LIN {X 0,Y 545.021,Z 219.093,A -85,B 0,C 180,E1 -3757.239,E2 -3757.239} C_VEL
LIN {X 0,Y 545.107,Z 219.079,A -85,B 0,C 180,E1 -3760.412,E2 -3760.412} C_VEL
LIN {X 0,Y 545.034,Z 219.089,A -85,B 0,C 180,E1 -3763.518,E2 -3763.518} C_VEL
LIN {X 0,Y 545.055,Z 219.086,A -85,B 0,C 180,E1 -3765.816,E2 -3765.816} C_VEL
LIN {X 0,Y 545.099,Z 219.082,A -85,B 0,C 180,E1 -3768.847,E2 -3768.847} C_VEL
LIN {X 0,Y 545.052,Z 219.085,A -85,B 0,C 180,E1 -3771.843,E2 -3771.843} C_VEL
LIN {X 0,Y 545.112,Z 219.078,A -85,B 0,C 180,E1 -3774.077,E2 -3774.077} C_VEL
LIN {X 0,Y 545.03,Z 219.094,A -85,B 0,C 180,E1 -3775.56,E2 -3775.56} C_VEL
LIN {X 0,Y 545.164,Z 219.076,A -85,B 0,C 180,E1 -3777.781,E2 -3777.781} C_VEL
LIN {X 0,Y 545.162,Z 219.073,A -85,B 0,C 180,E1 -3779.997,E2 -3779.997} C_VEL
LIN {X 0,Y 545.133,Z 219.076,A -85,B 0,C 180,E1 -3782.953,E2 -3782.953} C_VEL
LIN {X 0,Y 545.107,Z 219.084,A -85,B 0,C 180,E1 -3785.917,E2 -3785.917} C_VEL
LIN {X 0,Y 545.074,Z 219.082,A -85,B 0,C 180,E1 -3788.898,E2 -3788.898} C_VEL
LIN {X 0,Y 545.078,Z 219.091,A -85,B 0,C 180,E1 -3791.902,E2 -3791.902} C_VEL
LIN {X 0,Y 545.057,Z 219.085,A -85,B 0,C 180,E1 -3794.941,E2 -3794.941} C_VEL
LIN {X 0,Y 545.034,Z 219.097,A -85,B 0,C 180,E1 -3798.024,E2 -3798.024} C_VEL
LIN {X 0,Y 545.066,Z 219.089,A -85,B 0,C 180,E1 -3800.369,E2 -3800.369} C_VEL
LIN {X 0,Y 545.053,Z 219.086,A -85,B 0,C 180,E1 -3803.557,E2 -3803.557} C_VEL
LIN {X 0,Y 545.047,Z 219.091,A -85,B 0,C 180,E1 -3805.998,E2 -3805.998} C_VEL
LIN {X 0,Y 545.059,Z 219.086,A -85,B 0,C 180,E1 -3808.746,E2 -3808.746} C_VEL
LIN {X 0,Y 545.027,Z 219.089,A -85,B 0,C 180,E1 -3811.676,E2 -3811.676} C_VEL
LIN {X 0,Y 545.05,Z 219.094,A -85,B 0,C 180,E1 -3814.56,E2 -3814.56} C_VEL
LIN {X 0,Y 545.041,Z 219.091,A -85,B 0,C 180,E1 -3816.959,E2 -3816.959} C_VEL
LIN {X 0,Y 544.33,Z 219.178,A -85,B 0,C 180,E1 -3817.575,E2 -3817.575} C_VEL
LIN {X 0,Y 541.474,Z 219.539,A -85,B 0,C 180,E1 -3818.576,E2 -3818.576} C_VEL
LIN {X 0,Y 539.096,Z 219.831,A -85,B 0,C 180,E1 -3819.382,E2 -3819.382} C_VEL
LIN {X 0,Y 538.089,Z 219.955,A -85,B 0,C 180,E1 -3820.004,E2 -3820.004} C_VEL
LIN {X 0,Y 538.012,Z 219.965,A -85,B 0,C 180,E1 -3820.215,E2 -3820.215} C_VEL
LIN {X 0,Y 537.997,Z 219.971,A -85,B 0,C 180,E1 -3822.986,E2 -3822.986} C_VEL
LIN {X 0,Y 537.991,Z 219.968,A -85,B 0,C 180,E1 -3825.923,E2 -3825.923} C_VEL
LIN {X 0,Y 538.074,Z 220.022,A -85,B 0,C 180,E1 -3827.863,E2 -3827.863} C_VEL
LIN {X 0,Y 538.65,Z 224.83,A -85,B 0,C 180,E1 -3828.767,E2 -3828.767} C_VEL
LIN {X 0,Y 538.391,Z 241.013,A -85,B 0,C 180,E1 -3831.549,E2 -3831.549} C_VEL
LIN {X 0,Y 538.239,Z 257.087,A -85,B 0,C 180,E1 -3834.274,E2 -3834.274} C_VEL
LIN {X 0,Y 539.614,Z 265.361,A -85,B 0,C 180,E1 -3834.454,E2 -3834.454} C_VEL
LIN {X 0,Y 539.316,Z 364.892,A -85,B 0,C 180,E1 -3835.809,E2 -3835.809} C_VEL
LIN {X 0,Y 539.152,Z 377.977,A -85,B 0,C 180,E1 -3836.143,E2 -3836.143} C_VEL
LIN {X 0,Y 538.948,Z 391.003,A -85,B 0,C 180,E1 -3836.637,E2 -3836.637} C_VEL
LIN {X 0,Y 538.715,Z 402.354,A -85,B 0,C 180,E1 -3837.223,E2 -3837.223} C_VEL
LIN {X 0,Y 538.426,Z 414.542,A -85,B 0,C 180,E1 -3838.033,E2 -3838.033} C_VEL
LIN {X 0,Y 538.241,Z 425.418,A -85,B 0,C 180,E1 -3838.953,E2 -3838.953} C_VEL
LIN {X 0,Y 538.08,Z 433.702,A -85,B 0,C 180,E1 -3839.812,E2 -3839.812} C_VEL
LIN {X 0,Y 537.855,Z 442.133,A -85,B 0,C 180,E1 -3840.875,E2 -3840.875} C_VEL
LIN {X 0,Y 537.765,Z 448.984,A -85,B 0,C 180,E1 -3841.936,E2 -3841.936} C_VEL
LIN {X 0,Y 537.635,Z 455.498,A -85,B 0,C 180,E1 -3843.195,E2 -3843.195} C_VEL
LIN {X 0,Y 537.571,Z 460.422,A -85,B 0,C 180,E1 -3844.443,E2 -3844.443} C_VEL
LIN {X 0,Y 537.518,Z 464.02,A -85,B 0,C 180,E1 -3845.68,E2 -3845.68} C_VEL
LIN {X 0,Y 537.467,Z 466.427,A -85,B 0,C 180,E1 -3846.905,E2 -3846.905} C_VEL
LIN {X 0,Y 537.452,Z 467.776,A -85,B 0,C 180,E1 -3848.178,E2 -3848.178} C_VEL
LIN {X 0,Y 537.449,Z 468.012,A -85,B 0,C 180,E1 -3849.326,E2 -3849.326} C_VEL
LIN {X 0,Y 537.484,Z 467.525,A -85,B 0,C 180,E1 -3850.282,E2 -3850.282} C_VEL
LIN {X 0,Y 537.451,Z 465.527,A -85,B 0,C 180,E1 -3851.711,E2 -3851.711} C_VEL
LIN {X 0,Y 537.512,Z 463.492,A -85,B 0,C 180,E1 -3852.629,E2 -3852.629} C_VEL
LIN {X 0,Y 537.561,Z 460.326,A -85,B 0,C 180,E1 -3853.676,E2 -3853.676} C_VEL
LIN {X 0,Y 537.623,Z 455.716,A -85,B 0,C 180,E1 -3854.845,E2 -3854.845} C_VEL
LIN {X 0,Y 537.724,Z 449.838,A -85,B 0,C 180,E1 -3856.009,E2 -3856.009} C_VEL
LIN {X 0,Y 537.865,Z 442.467,A -85,B 0,C 180,E1 -3857.167,E2 -3857.167} C_VEL
LIN {X 0,Y 538.019,Z 433.799,A -85,B 0,C 180,E1 -3858.267,E2 -3858.267} C_VEL
LIN {X 0,Y 538.275,Z 423.895,A -85,B 0,C 180,E1 -3859.279,E2 -3859.279} C_VEL
LIN {X 0,Y 538.488,Z 413.423,A -85,B 0,C 180,E1 -3860.138,E2 -3860.138} C_VEL
LIN {X 0,Y 538.765,Z 401.776,A -85,B 0,C 180,E1 -3860.901,E2 -3860.901} C_VEL
LIN {X 0,Y 538.981,Z 389.466,A -85,B 0,C 180,E1 -3861.519,E2 -3861.519} C_VEL
LIN {X 0,Y 539.187,Z 375.978,A -85,B 0,C 180,E1 -3862.01,E2 -3862.01} C_VEL
LIN {X 0,Y 539.352,Z 363.101,A -85,B 0,C 180,E1 -3862.314,E2 -3862.314} C_VEL
LIN {X 0,Y 539.454,Z 264.301,A -85,B 0,C 180,E1 -3863.655,E2 -3863.655} C_VEL
LIN {X 0,Y 538.269,Z 257.585,A -85,B 0,C 180,E1 -3863.794,E2 -3863.794} C_VEL
LIN {X 0,Y 538.202,Z 256.454,A -85,B 0,C 180,E1 -3863.911,E2 -3863.911} C_VEL
LIN {X 0,Y 538.606,Z 238.795,A -85,B 0,C 180,E1 -3867.009,E2 -3867.009} C_VEL
LIN {X 0,Y 538.771,Z 224.137,A -85,B 0,C 180,E1 -3869.627,E2 -3869.627} C_VEL
LIN {X 0,Y 538.129,Z 220.013,A -85,B 0,C 180,E1 -3870.445,E2 -3870.445} C_VEL
LIN {X 0,Y 538.102,Z 219.959,A -85,B 0,C 180,E1 -3872.996,E2 -3872.996} C_VEL
LIN {X 0,Y 538.081,Z 219.957,A -85,B 0,C 180,E1 -3875.999,E2 -3875.999} C_VEL
LIN {X 0,Y 538.025,Z 219.962,A -85,B 0,C 180,E1 -3879.019,E2 -3879.019} C_VEL
LIN {X 0,Y 538.039,Z 219.961,A -85,B 0,C 180,E1 -3882.065,E2 -3882.065} C_VEL
LIN {X 0,Y 538,Z 219.965,A -85,B 0,C 180,E1 -3885.146,E2 -3885.146} C_VEL
LIN {X 0,Y 537.989,Z 219.968,A -85,B 0,C 180,E1 -3888.273,E2 -3888.273} C_VEL
LIN {X 0,Y 537.998,Z 219.964,A -85,B 0,C 180,E1 -3890.654,E2 -3890.654} C_VEL
LIN {X 0,Y 537.963,Z 219.976,A -85,B 0,C 180,E1 -3893.891,E2 -3893.891} C_VEL
LIN {X 0,Y 537.976,Z 219.971,A -85,B 0,C 180,E1 -3896.371,E2 -3896.371} C_VEL
LIN {X 0,Y 537.994,Z 219.964,A -85,B 0,C 180,E1 -3898.936,E2 -3898.936} C_VEL
LIN {X 0,Y 537.975,Z 219.97,A -85,B 0,C 180,E1 -3901.89,E2 -3901.89} C_VEL
LIN {X 0,Y 537.963,Z 219.973,A -85,B 0,C 180,E1 -3904.618,E2 -3904.618} C_VEL
LIN {X 0,Y 537.952,Z 219.971,A -85,B 0,C 180,E1 -3907.882,E2 -3907.882} C_VEL
LIN {X 0,Y 537.97,Z 219.973,A -85,B 0,C 180,E1 -3910.784,E2 -3910.784} C_VEL
LIN {X 0,Y 537.984,Z 219.967,A -85,B 0,C 180,E1 -3914.076,E2 -3914.076} C_VEL
LIN {X 0,Y 537.974,Z 219.972,A -85,B 0,C 180,E1 -3917.02,E2 -3917.02} C_VEL
LIN {X 0,Y 537.987,Z 219.966,A -85,B 0,C 180,E1 -3920.206,E2 -3920.206} C_VEL
LIN {X 0,Y 538.005,Z 219.971,A -85,B 0,C 180,E1 -3923.071,E2 -3923.071} C_VEL
LIN {X 0,Y 537.992,Z 219.964,A -85,B 0,C 180,E1 -3925.83,E2 -3925.83} C_VEL
LIN {X 0,Y 537.98,Z 219.967,A -85,B 0,C 180,E1 -3928.502,E2 -3928.502} C_VEL
LIN {X 0,Y 537.989,Z 219.973,A -85,B 0,C 180,E1 -3931.1,E2 -3931.1} C_VEL
LIN {X 0,Y 537.968,Z 219.972,A -85,B 0,C 180,E1 -3933.634,E2 -3933.634} C_VEL
LIN {X 0,Y 537.998,Z 219.964,A -85,B 0,C 180,E1 -3936.126,E2 -3936.126} C_VEL
LIN {X 0,Y 538.03,Z 219.967,A -85,B 0,C 180,E1 -3939.352,E2 -3939.352} C_VEL
LIN {X 0,Y 538.002,Z 219.97,A -85,B 0,C 180,E1 -3941.733,E2 -3941.733} C_VEL
LIN {X 0,Y 538.046,Z 219.96,A -85,B 0,C 180,E1 -3945.151,E2 -3945.151} C_VEL
LIN {X 0,Y 538.038,Z 219.959,A -85,B 0,C 180,E1 -3948.43,E2 -3948.43} C_VEL
LIN {X 0,Y 538.041,Z 219.966,A -85,B 0,C 180,E1 -3951.742,E2 -3951.742} C_VEL
LIN {X 0,Y 538.124,Z 219.948,A -85,B 0,C 180,E1 -3954.758,E2 -3954.758} C_VEL
LIN {X 0,Y 538.163,Z 219.948,A -85,B 0,C 180,E1 -3957.758,E2 -3957.758} C_VEL
LIN {X 0,Y 538.181,Z 219.942,A -85,B 0,C 180,E1 -3960.751,E2 -3960.751} C_VEL
LIN {X 0,Y 538.123,Z 219.948,A -85,B 0,C 180,E1 -3962.997,E2 -3962.997} C_VEL
LIN {X 0,Y 538.089,Z 219.956,A -85,B 0,C 180,E1 -3966,E2 -3966} C_VEL
LIN {X 0,Y 538.036,Z 219.96,A -85,B 0,C 180,E1 -3969.021,E2 -3969.021} C_VEL
LIN {X 0,Y 538.07,Z 219.957,A -85,B 0,C 180,E1 -3972.065,E2 -3972.065} C_VEL
LIN {X 0,Y 538.051,Z 219.959,A -85,B 0,C 180,E1 -3975.146,E2 -3975.146} C_VEL
LIN {X 0,Y 538.02,Z 219.963,A -85,B 0,C 180,E1 -3978.273,E2 -3978.273} C_VEL
LIN {X 0,Y 538.045,Z 219.965,A -85,B 0,C 180,E1 -3980.653,E2 -3980.653} C_VEL
LIN {X 0,Y 538.019,Z 219.961,A -85,B 0,C 180,E1 -3983.879,E2 -3983.879} C_VEL
LIN {X 0,Y 538.003,Z 219.964,A -85,B 0,C 180,E1 -3986.371,E2 -3986.371} C_VEL
LIN {X 0,Y 538.006,Z 219.97,A -85,B 0,C 180,E1 -3988.927,E2 -3988.927} C_VEL
LIN {X 0,Y 538.013,Z 219.962,A -85,B 0,C 180,E1 -3991.886,E2 -3991.886} C_VEL
LIN {X 0,Y 538.009,Z 219.963,A -85,B 0,C 180,E1 -3994.616,E2 -3994.616} C_VEL
LIN {X 0,Y 538.012,Z 219.968,A -85,B 0,C 180,E1 -3997.17,E2 -3997.17} C_VEL
LIN {X 0,Y 538.03,Z 219.964,A -85,B 0,C 180,E1 -3999.798,E2 -3999.798} C_VEL
LIN {X 0,Y 537.986,Z 219.965,A -85,B 0,C 180,E1 -4002.791,E2 -4002.791} C_VEL
LIN {X 0,Y 538.006,Z 219.965,A -85,B 0,C 180,E1 -4005.137,E2 -4005.137} C_VEL
LIN {X 0,Y 538.006,Z 219.965,A -85,B 0,C 180,E1 -4008.223,E2 -4008.223} C_VEL
LIN {X 0,Y 538.022,Z 219.962,A -85,B 0,C 180,E1 -4011.169,E2 -4011.169} C_VEL
LIN {X 0,Y 537.999,Z 219.971,A -85,B 0,C 180,E1 -4014.09,E2 -4014.09} C_VEL
LIN {X 0,Y 538.043,Z 219.958,A -85,B 0,C 180,E1 -4016.727,E2 -4016.727} C_VEL
LIN {X 0,Y 538.017,Z 219.963,A -85,B 0,C 180,E1 -4019.56,E2 -4019.56} C_VEL
LIN {X 0,Y 538.03,Z 219.968,A -85,B 0,C 180,E1 -4021.949,E2 -4021.949} C_VEL
LIN {X 0,Y 538.04,Z 219.968,A -85,B 0,C 180,E1 -4024.465,E2 -4024.465} C_VEL
LIN {X 0,Y 538.066,Z 220.043,A -85,B 0,C 180,E1 -4026.879,E2 -4026.879} C_VEL
LIN {X 0,Y 539.068,Z 225.745,A -85,B 0,C 180,E1 -4027.92,E2 -4027.92} C_VEL
LIN {X 0,Y 538.843,Z 239.465,A -85,B 0,C 180,E1 -4030.176,E2 -4030.176} C_VEL
LIN {X 0,Y 538.581,Z 255.211,A -85,B 0,C 180,E1 -4032.729,E2 -4032.729} C_VEL
LIN {X 0,Y 538.326,Z 271.075,A -85,B 0,C 180,E1 -4035.23,E2 -4035.23} C_VEL
LIN {X 0,Y 539.67,Z 279.984,A -85,B 0,C 180,E1 -4035.412,E2 -4035.412} C_VEL
LIN {X 0,Y 539.334,Z 378.53,A -85,B 0,C 180,E1 -4036.745,E2 -4036.745} C_VEL
LIN {X 0,Y 539.178,Z 391.879,A -85,B 0,C 180,E1 -4037.077,E2 -4037.077} C_VEL
LIN {X 0,Y 538.939,Z 404.075,A -85,B 0,C 180,E1 -4037.526,E2 -4037.526} C_VEL
LIN {X 0,Y 538.758,Z 415.668,A -85,B 0,C 180,E1 -4038.101,E2 -4038.101} C_VEL
LIN {X 0,Y 538.552,Z 426.682,A -85,B 0,C 180,E1 -4038.806,E2 -4038.806} C_VEL
LIN {X 0,Y 538.253,Z 437.345,A -85,B 0,C 180,E1 -4039.656,E2 -4039.656} C_VEL
LIN {X 0,Y 538.07,Z 446.95,A -85,B 0,C 180,E1 -4040.602,E2 -4040.602} C_VEL
LIN {X 0,Y 537.915,Z 454.822,A -85,B 0,C 180,E1 -4041.547,E2 -4041.547} C_VEL
LIN {X 0,Y 537.758,Z 462.507,A -85,B 0,C 180,E1 -4042.678,E2 -4042.678} C_VEL
LIN {X 0,Y 537.697,Z 469.588,A -85,B 0,C 180,E1 -4043.997,E2 -4043.997} C_VEL
LIN {X 0,Y 537.541,Z 474.296,A -85,B 0,C 180,E1 -4045.124,E2 -4045.124} C_VEL
LIN {X 0,Y 537.592,Z 477.894,A -85,B 0,C 180,E1 -4046.251,E2 -4046.251} C_VEL
LIN {X 0,Y 537.552,Z 479.749,A -85,B 0,C 180,E1 -4047.001,E2 -4047.001} C_VEL
LIN {X 0,Y 537.451,Z 482.132,A -85,B 0,C 180,E1 -4048.5,E2 -4048.5} C_VEL
LIN {X 0,Y 537.442,Z 482.954,A -85,B 0,C 180,E1 -4049.999,E2 -4049.999} C_VEL
LIN {X 0,Y 537.451,Z 482.136,A -85,B 0,C 180,E1 -4051.497,E2 -4051.497} C_VEL
LIN {X 0,Y 537.552,Z 479.757,A -85,B 0,C 180,E1 -4052.997,E2 -4052.997} C_VEL
LIN {X 0,Y 537.604,Z 476.834,A -85,B 0,C 180,E1 -4054.122,E2 -4054.122} C_VEL
LIN {X 0,Y 537.588,Z 472.874,A -85,B 0,C 180,E1 -4055.249,E2 -4055.249} C_VEL
LIN {X 0,Y 537.642,Z 468.042,A -85,B 0,C 180,E1 -4056.324,E2 -4056.324} C_VEL
LIN {X 0,Y 537.773,Z 461.359,A -85,B 0,C 180,E1 -4057.508,E2 -4057.508} C_VEL
LIN {X 0,Y 537.933,Z 453.348,A -85,B 0,C 180,E1 -4058.64,E2 -4058.64} C_VEL
LIN {X 0,Y 538.115,Z 445.182,A -85,B 0,C 180,E1 -4059.584,E2 -4059.584} C_VEL
LIN {X 0,Y 538.333,Z 435.22,A -85,B 0,C 180,E1 -4060.53,E2 -4060.53} C_VEL
LIN {X 0,Y 538.589,Z 425.392,A -85,B 0,C 180,E1 -4061.286,E2 -4061.286} C_VEL
LIN {X 0,Y 538.759,Z 414.935,A -85,B 0,C 180,E1 -4061.938,E2 -4061.938} C_VEL
LIN {X 0,Y 538.952,Z 401.845,A -85,B 0,C 180,E1 -4062.567,E2 -4062.567} C_VEL
LIN {X 0,Y 539.19,Z 388.79,A -85,B 0,C 180,E1 -4063.016,E2 -4063.016} C_VEL
LIN {X 0,Y 539.334,Z 375.751,A -85,B 0,C 180,E1 -4063.3,E2 -4063.3} C_VEL
LIN {X 0,Y 539.571,Z 279.118,A -85,B 0,C 180,E1 -4064.601,E2 -4064.601} C_VEL
LIN {X 0,Y 538.312,Z 271.159,A -85,B 0,C 180,E1 -4064.763,E2 -4064.763} C_VEL
LIN {X 0,Y 538.31,Z 267.291,A -85,B 0,C 180,E1 -4065.329,E2 -4065.329} C_VEL
LIN {X 0,Y 538.645,Z 249.049,A -85,B 0,C 180,E1 -4068.247,E2 -4068.247} C_VEL
LIN {X 0,Y 539.017,Z 230.767,A -85,B 0,C 180,E1 -4071.211,E2 -4071.211} C_VEL
LIN {X 0,Y 538.89,Z 224.65,A -85,B 0,C 180,E1 -4072.221,E2 -4072.221} C_VEL
LIN {X 0,Y 538.04,Z 220.032,A -85,B 0,C 180,E1 -4073.069,E2 -4073.069} C_VEL
LIN {X 0,Y 538.041,Z 219.963,A -85,B 0,C 180,E1 -4076.365,E2 -4076.365} C_VEL
LIN {X 0,Y 538.031,Z 219.961,A -85,B 0,C 180,E1 -4078.932,E2 -4078.932} C_VEL
LIN {X 0,Y 538.011,Z 219.972,A -85,B 0,C 180,E1 -4081.885,E2 -4081.885} C_VEL
LIN {X 0,Y 538.01,Z 219.963,A -85,B 0,C 180,E1 -4084.615,E2 -4084.615} C_VEL
LIN {X 0,Y 537.998,Z 219.965,A -85,B 0,C 180,E1 -4087.167,E2 -4087.167} C_VEL
LIN {X 0,Y 538.009,Z 219.967,A -85,B 0,C 180,E1 -4089.796,E2 -4089.796} C_VEL
LIN {X 0,Y 538.018,Z 219.966,A -85,B 0,C 180,E1 -4091.875,E2 -4091.875} C_VEL
LIN {X 0,Y 538.002,Z 219.965,A -85,B 0,C 180,E1 -4094.861,E2 -4094.861} C_VEL
LIN {X 0,Y 537.997,Z 219.961,A -85,B 0,C 180,E1 -4097.21,E2 -4097.21} C_VEL
LIN {X 0,Y 538.007,Z 219.97,A -85,B 0,C 180,E1 -4100.2,E2 -4100.2} C_VEL
LIN {X 0,Y 538.014,Z 219.963,A -85,B 0,C 180,E1 -4103.064,E2 -4103.064} C_VEL
LIN {X 0,Y 538.012,Z 219.963,A -85,B 0,C 180,E1 -4105.824,E2 -4105.824} C_VEL
LIN {X 0,Y 538.003,Z 219.97,A -85,B 0,C 180,E1 -4108.496,E2 -4108.496} C_VEL
LIN {X 0,Y 538.013,Z 219.966,A -85,B 0,C 180,E1 -4111.095,E2 -4111.095} C_VEL
LIN {X 0,Y 537.987,Z 219.965,A -85,B 0,C 180,E1 -4113.628,E2 -4113.628} C_VEL
LIN {X 0,Y 538,Z 219.964,A -85,B 0,C 180,E1 -4116.12,E2 -4116.12} C_VEL
LIN {X 0,Y 538.025,Z 219.964,A -85,B 0,C 180,E1 -4119.346,E2 -4119.346} C_VEL
LIN {X 0,Y 538.028,Z 219.961,A -85,B 0,C 180,E1 -4122.465,E2 -4122.465} C_VEL
LIN {X 0,Y 538.028,Z 219.963,A -85,B 0,C 180,E1 -4125.627,E2 -4125.627} C_VEL
LIN {X 0,Y 538.061,Z 219.956,A -85,B 0,C 180,E1 -4128.699,E2 -4128.699} C_VEL
LIN {X 0,Y 538.021,Z 219.961,A -85,B 0,C 180,E1 -4131.736,E2 -4131.736} C_VEL
LIN {X 0,Y 538.069,Z 219.956,A -85,B 0,C 180,E1 -4133.999,E2 -4133.999} C_VEL
LIN {X 0,Y 537.997,Z 219.971,A -85,B 0,C 180,E1 -4135.502,E2 -4135.502} C_VEL
LIN {X 0,Y 538.137,Z 219.952,A -85,B 0,C 180,E1 -4137.752,E2 -4137.752} C_VEL
LIN {X 0,Y 538.132,Z 219.949,A -85,B 0,C 180,E1 -4139.997,E2 -4139.997} C_VEL
LIN {X 0,Y 538.101,Z 219.952,A -85,B 0,C 180,E1 -4142.992,E2 -4142.992} C_VEL
LIN {X 0,Y 538.062,Z 219.961,A -85,B 0,C 180,E1 -4145.995,E2 -4145.995} C_VEL
LIN {X 0,Y 538.027,Z 219.96,A -85,B 0,C 180,E1 -4149.015,E2 -4149.015} C_VEL
LIN {X 0,Y 538.037,Z 219.965,A -85,B 0,C 180,E1 -4152.06,E2 -4152.06} C_VEL
LIN {X 0,Y 538.017,Z 219.962,A -85,B 0,C 180,E1 -4155.141,E2 -4155.141} C_VEL
LIN {X 0,Y 537.987,Z 219.971,A -85,B 0,C 180,E1 -4158.268,E2 -4158.268} C_VEL
LIN {X 0,Y 538.011,Z 219.965,A -85,B 0,C 180,E1 -4160.649,E2 -4160.649} C_VEL
LIN {X 0,Y 537.975,Z 219.972,A -85,B 0,C 180,E1 -4163.886,E2 -4163.886} C_VEL
LIN {X 0,Y 538.009,Z 219.971,A -85,B 0,C 180,E1 -4166.364,E2 -4166.364} C_VEL
LIN {X 0,Y 538,Z 219.964,A -85,B 0,C 180,E1 -4168.931,E2 -4168.931} C_VEL
LIN {X 0,Y 537.982,Z 219.968,A -85,B 0,C 180,E1 -4171.885,E2 -4171.885} C_VEL
LIN {X 0,Y 538,Z 219.971,A -85,B 0,C 180,E1 -4174.618,E2 -4174.618} C_VEL
LIN {X 0,Y 537.977,Z 219.969,A -85,B 0,C 180,E1 -4177.169,E2 -4177.169} C_VEL
LIN {X 0,Y 538.012,Z 219.965,A -85,B 0,C 180,E1 -4180.215,E2 -4180.215} C_VEL
LIN {X 0,Y 537.358,Z 220.052,A -85,B 0,C 180,E1 -4180.84,E2 -4180.84} C_VEL
LIN {X 0,Y 534.502,Z 220.407,A -85,B 0,C 180,E1 -4181.854,E2 -4181.854} C_VEL
LIN {X 0,Y 532.072,Z 220.711,A -85,B 0,C 180,E1 -4182.671,E2 -4182.671} C_VEL
LIN {X 0,Y 531.019,Z 220.837,A -85,B 0,C 180,E1 -4183.302,E2 -4183.302} C_VEL
LIN {X 0,Y 530.929,Z 220.847,A -85,B 0,C 180,E1 -4183.516,E2 -4183.516} C_VEL
LIN {X 0,Y 530.931,Z 220.852,A -85,B 0,C 180,E1 -4186.504,E2 -4186.504} C_VEL
LIN {X 0,Y 531.014,Z 220.926,A -85,B 0,C 180,E1 -4187.755,E2 -4187.755} C_VEL
LIN {X 0,Y 531.668,Z 225.543,A -85,B 0,C 180,E1 -4188.631,E2 -4188.631} C_VEL
LIN {X 0,Y 531.45,Z 240.749,A -85,B 0,C 180,E1 -4191.274,E2 -4191.274} C_VEL
LIN {X 0,Y 531.224,Z 257.112,A -85,B 0,C 180,E1 -4194.07,E2 -4194.07} C_VEL
LIN {X 0,Y 532.148,Z 262.625,A -85,B 0,C 180,E1 -4194.206,E2 -4194.206} C_VEL
LIN {X 0,Y 532.79,Z 267.89,A -85,B 0,C 180,E1 -4194.297,E2 -4194.297} C_VEL
LIN {X 0,Y 532.415,Z 364.859,A -85,B 0,C 180,E1 -4195.633,E2 -4195.633} C_VEL
LIN {X 0,Y 532.227,Z 378.628,A -85,B 0,C 180,E1 -4195.991,E2 -4195.991} C_VEL
LIN {X 0,Y 532.03,Z 390.825,A -85,B 0,C 180,E1 -4196.462,E2 -4196.462} C_VEL
LIN {X 0,Y 531.757,Z 402.623,A -85,B 0,C 180,E1 -4197.077,E2 -4197.077} C_VEL
LIN {X 0,Y 531.479,Z 414.472,A -85,B 0,C 180,E1 -4197.876,E2 -4197.876} C_VEL
LIN {X 0,Y 531.262,Z 424.493,A -85,B 0,C 180,E1 -4198.721,E2 -4198.721} C_VEL
LIN {X 0,Y 531.034,Z 433.441,A -85,B 0,C 180,E1 -4199.647,E2 -4199.647} C_VEL
LIN {X 0,Y 530.825,Z 441.541,A -85,B 0,C 180,E1 -4200.67,E2 -4200.67} C_VEL
LIN {X 0,Y 530.702,Z 449.768,A -85,B 0,C 180,E1 -4201.96,E2 -4201.96} C_VEL
LIN {X 0,Y 530.546,Z 456.091,A -85,B 0,C 180,E1 -4203.233,E2 -4203.233} C_VEL
LIN {X 0,Y 530.48,Z 461.198,A -85,B 0,C 180,E1 -4204.59,E2 -4204.59} C_VEL
LIN {X 0,Y 530.44,Z 464.389,A -85,B 0,C 180,E1 -4205.751,E2 -4205.751} C_VEL
LIN {X 0,Y 530.397,Z 466.074,A -85,B 0,C 180,E1 -4206.579,E2 -4206.579} C_VEL
LIN {X 0,Y 530.352,Z 467.803,A -85,B 0,C 180,E1 -4208.052,E2 -4208.052} C_VEL
LIN {X 0,Y 530.338,Z 468.164,A -85,B 0,C 180,E1 -4209.036,E2 -4209.036} C_VEL
LIN {X 0,Y 530.391,Z 467.717,A -85,B 0,C 180,E1 -4210.17,E2 -4210.17} C_VEL
LIN {X 0,Y 530.363,Z 466.16,A -85,B 0,C 180,E1 -4211.458,E2 -4211.458} C_VEL
LIN {X 0,Y 530.401,Z 463.911,A -85,B 0,C 180,E1 -4212.542,E2 -4212.542} C_VEL
LIN {X 0,Y 530.482,Z 460.057,A -85,B 0,C 180,E1 -4213.848,E2 -4213.848} C_VEL
LIN {X 0,Y 530.601,Z 454.528,A -85,B 0,C 180,E1 -4215.199,E2 -4215.199} C_VEL
LIN {X 0,Y 530.712,Z 448.155,A -85,B 0,C 180,E1 -4216.406,E2 -4216.406} C_VEL
LIN {X 0,Y 530.869,Z 440.409,A -85,B 0,C 180,E1 -4217.578,E2 -4217.578} C_VEL
LIN {X 0,Y 531.023,Z 432.484,A -85,B 0,C 180,E1 -4218.551,E2 -4218.551} C_VEL
LIN {X 0,Y 531.284,Z 422.795,A -85,B 0,C 180,E1 -4219.521,E2 -4219.521} C_VEL
LIN {X 0,Y 531.524,Z 412.077,A -85,B 0,C 180,E1 -4220.392,E2 -4220.392} C_VEL
LIN {X 0,Y 531.81,Z 401.681,A -85,B 0,C 180,E1 -4221.068,E2 -4221.068} C_VEL
LIN {X 0,Y 532.029,Z 390.415,A -85,B 0,C 180,E1 -4221.646,E2 -4221.646} C_VEL
LIN {X 0,Y 532.257,Z 377.021,A -85,B 0,C 180,E1 -4222.15,E2 -4222.15} C_VEL
LIN {X 0,Y 532.448,Z 364.482,A -85,B 0,C 180,E1 -4222.464,E2 -4222.464} C_VEL
LIN {X 0,Y 532.614,Z 265.242,A -85,B 0,C 180,E1 -4223.835,E2 -4223.835} C_VEL
LIN {X 0,Y 531.246,Z 257.568,A -85,B 0,C 180,E1 -4223.997,E2 -4223.997} C_VEL
LIN {X 0,Y 531.215,Z 256.505,A -85,B 0,C 180,E1 -4224.116,E2 -4224.116} C_VEL
LIN {X 0,Y 531.634,Z 238.325,A -85,B 0,C 180,E1 -4227.349,E2 -4227.349} C_VEL
LIN {X 0,Y 531.837,Z 225.744,A -85,B 0,C 180,E1 -4229.623,E2 -4229.623} C_VEL
LIN {X 0,Y 531.108,Z 220.878,A -85,B 0,C 180,E1 -4230.594,E2 -4230.594} C_VEL
LIN {X 0,Y 531.068,Z 220.836,A -85,B 0,C 180,E1 -4233.036,E2 -4233.036} C_VEL
LIN {X 0,Y 531.036,Z 220.834,A -85,B 0,C 180,E1 -4236.079,E2 -4236.079} C_VEL
LIN {X 0,Y 530.986,Z 220.841,A -85,B 0,C 180,E1 -4239.14,E2 -4239.14} C_VEL
LIN {X 0,Y 530.997,Z 220.837,A -85,B 0,C 180,E1 -4242.227,E2 -4242.227} C_VEL
LIN {X 0,Y 530.95,Z 220.845,A -85,B 0,C 180,E1 -4245.352,E2 -4245.352} C_VEL
LIN {X 0,Y 530.948,Z 220.842,A -85,B 0,C 180,E1 -4248.524,E2 -4248.524} C_VEL
LIN {X 0,Y 530.959,Z 220.84,A -85,B 0,C 180,E1 -4250.941,E2 -4250.941} C_VEL
LIN {X 0,Y 530.923,Z 220.851,A -85,B 0,C 180,E1 -4254.228,E2 -4254.228} C_VEL
LIN {X 0,Y 530.931,Z 220.845,A -85,B 0,C 180,E1 -4256.749,E2 -4256.749} C_VEL
LIN {X 0,Y 530.945,Z 220.842,A -85,B 0,C 180,E1 -4259.326,E2 -4259.326} C_VEL
LIN {X 0,Y 530.93,Z 220.851,A -85,B 0,C 180,E1 -4262.103,E2 -4262.103} C_VEL
LIN {X 0,Y 530.924,Z 220.847,A -85,B 0,C 180,E1 -4264.852,E2 -4264.852} C_VEL
LIN {X 0,Y 530.905,Z 220.847,A -85,B 0,C 180,E1 -4267.514,E2 -4267.514} C_VEL
LIN {X 0,Y 530.918,Z 220.854,A -85,B 0,C 180,E1 -4270.44,E2 -4270.44} C_VEL
LIN {X 0,Y 530.911,Z 220.846,A -85,B 0,C 180,E1 -4273.501,E2 -4273.501} C_VEL
LIN {X 0,Y 530.92,Z 220.851,A -85,B 0,C 180,E1 -4276.507,E2 -4276.507} C_VEL
LIN {X 0,Y 530.929,Z 220.845,A -85,B 0,C 180,E1 -4279.568,E2 -4279.568} C_VEL
LIN {X 0,Y 530.948,Z 220.846,A -85,B 0,C 180,E1 -4282.581,E2 -4282.581} C_VEL
LIN {X 0,Y 530.962,Z 220.845,A -85,B 0,C 180,E1 -4285.313,E2 -4285.313} C_VEL
LIN {X 0,Y 530.942,Z 220.842,A -85,B 0,C 180,E1 -4288.035,E2 -4288.035} C_VEL
LIN {X 0,Y 530.95,Z 220.846,A -85,B 0,C 180,E1 -4290.883,E2 -4290.883} C_VEL
LIN {X 0,Y 530.935,Z 220.853,A -85,B 0,C 180,E1 -4293.257,E2 -4293.257} C_VEL
LIN {X 0,Y 530.944,Z 220.844,A -85,B 0,C 180,E1 -4295.973,E2 -4295.973} C_VEL
LIN {X 0,Y 530.991,Z 220.84,A -85,B 0,C 180,E1 -4299.066,E2 -4299.066} C_VEL
LIN {X 0,Y 530.964,Z 220.849,A -85,B 0,C 180,E1 -4301.482,E2 -4301.482} C_VEL
LIN {X 0,Y 530.981,Z 220.837,A -85,B 0,C 180,E1 -4304.654,E2 -4304.654} C_VEL
LIN {X 0,Y 531.013,Z 220.844,A -85,B 0,C 180,E1 -4307.778,E2 -4307.778} C_VEL
LIN {X 0,Y 531.006,Z 220.834,A -85,B 0,C 180,E1 -4310.865,E2 -4310.865} C_VEL
LIN {X 0,Y 531.041,Z 220.84,A -85,B 0,C 180,E1 -4313.926,E2 -4313.926} C_VEL
LIN {X 0,Y 531.059,Z 220.828,A -85,B 0,C 180,E1 -4316.969,E2 -4316.969} C_VEL
LIN {X 0,Y 531.028,Z 220.836,A -85,B 0,C 180,E1 -4318.486,E2 -4318.486} C_VEL
LIN {X 0,Y 531.152,Z 220.818,A -85,B 0,C 180,E1 -4320.761,E2 -4320.761} C_VEL
LIN {X 0,Y 531.063,Z 220.828,A -85,B 0,C 180,E1 -4323.037,E2 -4323.037} C_VEL
LIN {X 0,Y 531.049,Z 220.834,A -85,B 0,C 180,E1 -4326.08,E2 -4326.08} C_VEL
LIN {X 0,Y 531.002,Z 220.836,A -85,B 0,C 180,E1 -4329.141,E2 -4329.141} C_VEL
LIN {X 0,Y 531.058,Z 220.828,A -85,B 0,C 180,E1 -4331.671,E2 -4331.671} C_VEL
LIN {X 0,Y 531.032,Z 220.836,A -85,B 0,C 180,E1 -4334.953,E2 -4334.953} C_VEL
LIN {X 0,Y 530.992,Z 220.836,A -85,B 0,C 180,E1 -4337.726,E2 -4337.726} C_VEL
LIN {X 0,Y 531.027,Z 220.833,A -85,B 0,C 180,E1 -4340.129,E2 -4340.129} C_VEL
LIN {X 0,Y 530.953,Z 220.846,A -85,B 0,C 180,E1 -4342.575,E2 -4342.575} C_VEL
LIN {X 0,Y 530.961,Z 220.849,A -85,B 0,C 180,E1 -4345.062,E2 -4345.062} C_VEL
LIN {X 0,Y 530.973,Z 220.841,A -85,B 0,C 180,E1 -4347.6,E2 -4347.6} C_VEL
LIN {X 0,Y 530.97,Z 220.841,A -85,B 0,C 180,E1 -4350.643,E2 -4350.643} C_VEL
LIN {X 0,Y 530.974,Z 220.844,A -85,B 0,C 180,E1 -4353.5,E2 -4353.5} C_VEL
LIN {X 0,Y 530.957,Z 220.841,A -85,B 0,C 180,E1 -4356.56,E2 -4356.56} C_VEL
LIN {X 0,Y 530.995,Z 220.846,A -85,B 0,C 180,E1 -4359.445,E2 -4359.445} C_VEL
LIN {X 0,Y 530.931,Z 220.844,A -85,B 0,C 180,E1 -4362.463,E2 -4362.463} C_VEL
LIN {X 0,Y 530.976,Z 220.845,A -85,B 0,C 180,E1 -4365.451,E2 -4365.451} C_VEL
LIN {X 0,Y 530.971,Z 220.839,A -85,B 0,C 180,E1 -4368.561,E2 -4368.561} C_VEL
LIN {X 0,Y 530.965,Z 220.845,A -85,B 0,C 180,E1 -4371.529,E2 -4371.529} C_VEL
LIN {X 0,Y 530.96,Z 220.843,A -85,B 0,C 180,E1 -4374.379,E2 -4374.379} C_VEL
LIN {X 0,Y 530.979,Z 220.838,A -85,B 0,C 180,E1 -4377.133,E2 -4377.133} C_VEL
LIN {X 0,Y 530.964,Z 220.845,A -85,B 0,C 180,E1 -4379.802,E2 -4379.802} C_VEL
LIN {X 0,Y 530.986,Z 220.845,A -85,B 0,C 180,E1 -4382.475,E2 -4382.475} C_VEL
LIN {X 0,Y 530.966,Z 220.845,A -85,B 0,C 180,E1 -4384.939,E2 -4384.939} C_VEL
LIN {X 0,Y 531.021,Z 221.038,A -85,B 0,C 180,E1 -4386.76,E2 -4386.76} C_VEL
LIN {X 0,Y 532.14,Z 227.81,A -85,B 0,C 180,E1 -4387.978,E2 -4387.978} C_VEL
LIN {X 0,Y 531.79,Z 244.228,A -85,B 0,C 180,E1 -4390.706,E2 -4390.706} C_VEL
LIN {X 0,Y 531.459,Z 259.97,A -85,B 0,C 180,E1 -4393.283,E2 -4393.283} C_VEL
LIN {X 0,Y 531.331,Z 270.933,A -85,B 0,C 180,E1 -4395.028,E2 -4395.028} C_VEL
LIN {X 0,Y 532.81,Z 280.939,A -85,B 0,C 180,E1 -4395.235,E2 -4395.235} C_VEL
LIN {X 0,Y 532.445,Z 378.366,A -85,B 0,C 180,E1 -4396.571,E2 -4396.571} C_VEL
LIN {X 0,Y 532.278,Z 391.739,A -85,B 0,C 180,E1 -4396.906,E2 -4396.906} C_VEL
LIN {X 0,Y 531.989,Z 403.945,A -85,B 0,C 180,E1 -4397.36,E2 -4397.36} C_VEL
LIN {X 0,Y 531.803,Z 415.6,A -85,B 0,C 180,E1 -4397.946,E2 -4397.946} C_VEL
LIN {X 0,Y 531.566,Z 426.566,A -85,B 0,C 180,E1 -4398.657,E2 -4398.657} C_VEL
LIN {X 0,Y 531.26,Z 437.233,A -85,B 0,C 180,E1 -4399.519,E2 -4399.519} C_VEL
LIN {X 0,Y 531.049,Z 446.841,A -85,B 0,C 180,E1 -4400.477,E2 -4400.477} C_VEL
LIN {X 0,Y 530.867,Z 454.715,A -85,B 0,C 180,E1 -4401.434,E2 -4401.434} C_VEL
LIN {X 0,Y 530.679,Z 462.402,A -85,B 0,C 180,E1 -4402.58,E2 -4402.58} C_VEL
LIN {X 0,Y 530.607,Z 469.485,A -85,B 0,C 180,E1 -4403.916,E2 -4403.916} C_VEL
LIN {X 0,Y 530.46,Z 474.195,A -85,B 0,C 180,E1 -4405.059,E2 -4405.059} C_VEL
LIN {X 0,Y 530.517,Z 477.795,A -85,B 0,C 180,E1 -4406.201,E2 -4406.201} C_VEL
LIN {X 0,Y 530.458,Z 479.65,A -85,B 0,C 180,E1 -4406.961,E2 -4406.961} C_VEL
LIN {X 0,Y 530.411,Z 481.041,A -85,B 0,C 180,E1 -4407.721,E2 -4407.721} C_VEL
LIN {X 0,Y 530.344,Z 482.64,A -85,B 0,C 180,E1 -4409.24,E2 -4409.24} C_VEL
LIN {X 0,Y 530.343,Z 482.856,A -85,B 0,C 180,E1 -4409.999,E2 -4409.999} C_VEL
LIN {X 0,Y 530.361,Z 482.037,A -85,B 0,C 180,E1 -4411.517,E2 -4411.517} C_VEL
LIN {X 0,Y 530.411,Z 481.047,A -85,B 0,C 180,E1 -4412.277,E2 -4412.277} C_VEL
LIN {X 0,Y 530.458,Z 479.657,A -85,B 0,C 180,E1 -4413.037,E2 -4413.037} C_VEL
LIN {X 0,Y 530.523,Z 476.732,A -85,B 0,C 180,E1 -4414.177,E2 -4414.177} C_VEL
LIN {X 0,Y 530.525,Z 472.771,A -85,B 0,C 180,E1 -4415.319,E2 -4415.319} C_VEL
LIN {X 0,Y 530.561,Z 467.272,A -85,B 0,C 180,E1 -4416.542,E2 -4416.542} C_VEL
LIN {X 0,Y 530.725,Z 460.016,A -85,B 0,C 180,E1 -4417.8,E2 -4417.8} C_VEL
LIN {X 0,Y 530.895,Z 451.747,A -85,B 0,C 180,E1 -4418.947,E2 -4418.947} C_VEL
LIN {X 0,Y 531.118,Z 443.268,A -85,B 0,C 180,E1 -4419.904,E2 -4419.904} C_VEL
LIN {X 0,Y 531.372,Z 432.788,A -85,B 0,C 180,E1 -4420.862,E2 -4420.862} C_VEL
LIN {X 0,Y 531.659,Z 421.868,A -85,B 0,C 180,E1 -4421.666,E2 -4421.666} C_VEL
LIN {X 0,Y 531.922,Z 411.042,A -85,B 0,C 180,E1 -4422.3,E2 -4422.3} C_VEL
LIN {X 0,Y 532.108,Z 399.356,A -85,B 0,C 180,E1 -4422.829,E2 -4422.829} C_VEL
LIN {X 0,Y 532.296,Z 385.885,A -85,B 0,C 180,E1 -4423.261,E2 -4423.261} C_VEL
LIN {X 0,Y 532.464,Z 372.519,A -85,B 0,C 180,E1 -4423.524,E2 -4423.524} C_VEL
LIN {X 0,Y 532.716,Z 280.048,A -85,B 0,C 180,E1 -4424.779,E2 -4424.779} C_VEL
LIN {X 0,Y 531.307,Z 270.886,A -85,B 0,C 180,E1 -4424.973,E2 -4424.973} C_VEL
LIN {X 0,Y 531.684,Z 251.272,A -85,B 0,C 180,E1 -4428.11,E2 -4428.11} C_VEL
LIN {X 0,Y 532.061,Z 231.854,A -85,B 0,C 180,E1 -4431.298,E2 -4431.298} C_VEL
LIN {X 0,Y 531.878,Z 225.67,A -85,B 0,C 180,E1 -4432.337,E2 -4432.337} C_VEL
LIN {X 0,Y 531.007,Z 220.939,A -85,B 0,C 180,E1 -4433.212,E2 -4433.212} C_VEL
LIN {X 0,Y 530.982,Z 220.846,A -85,B 0,C 180,E1 -4435.897,E2 -4435.897} C_VEL
LIN {X 0,Y 530.976,Z 220.841,A -85,B 0,C 180,E1 -4438.455,E2 -4438.455} C_VEL
LIN {X 0,Y 530.955,Z 220.842,A -85,B 0,C 180,E1 -4441.078,E2 -4441.078} C_VEL
LIN {X 0,Y 530.987,Z 220.844,A -85,B 0,C 180,E1 -4443.771,E2 -4443.771} C_VEL
LIN {X 0,Y 530.95,Z 220.845,A -85,B 0,C 180,E1 -4446.557,E2 -4446.557} C_VEL
LIN {X 0,Y 530.97,Z 220.84,A -85,B 0,C 180,E1 -4449.443,E2 -4449.443} C_VEL
LIN {X 0,Y 530.964,Z 220.845,A -85,B 0,C 180,E1 -4452.456,E2 -4452.456} C_VEL
LIN {X 0,Y 530.974,Z 220.84,A -85,B 0,C 180,E1 -4455.62,E2 -4455.62} C_VEL
LIN {X 0,Y 530.978,Z 220.846,A -85,B 0,C 180,E1 -4458.561,E2 -4458.561} C_VEL
LIN {X 0,Y 530.949,Z 220.842,A -85,B 0,C 180,E1 -4461.527,E2 -4461.527} C_VEL
LIN {X 0,Y 530.946,Z 220.849,A -85,B 0,C 180,E1 -4464.377,E2 -4464.377} C_VEL
LIN {X 0,Y 530.962,Z 220.842,A -85,B 0,C 180,E1 -4467.131,E2 -4467.131} C_VEL
LIN {X 0,Y 530.947,Z 220.842,A -85,B 0,C 180,E1 -4469.8,E2 -4469.8} C_VEL
LIN {X 0,Y 530.961,Z 220.845,A -85,B 0,C 180,E1 -4472.475,E2 -4472.475} C_VEL
LIN {X 0,Y 530.943,Z 220.85,A -85,B 0,C 180,E1 -4474.937,E2 -4474.937} C_VEL
LIN {X 0,Y 530.969,Z 220.839,A -85,B 0,C 180,E1 -4477.896,E2 -4477.896} C_VEL
LIN {X 0,Y 530.973,Z 220.843,A -85,B 0,C 180,E1 -4480.674,E2 -4480.674} C_VEL
LIN {X 0,Y 530.95,Z 220.849,A -85,B 0,C 180,E1 -4483.067,E2 -4483.067} C_VEL
LIN {X 0,Y 530.989,Z 220.842,A -85,B 0,C 180,E1 -4485.433,E2 -4485.433} C_VEL
LIN {X 0,Y 531.02,Z 220.832,A -85,B 0,C 180,E1 -4488.547,E2 -4488.547} C_VEL
LIN {X 0,Y 530.97,Z 220.841,A -85,B 0,C 180,E1 -4491.625,E2 -4491.625} C_VEL
LIN {X 0,Y 531.03,Z 220.834,A -85,B 0,C 180,E1 -4493.92,E2 -4493.92} C_VEL
LIN {X 0,Y 530.965,Z 220.848,A -85,B 0,C 180,E1 -4495.442,E2 -4495.442} C_VEL
LIN {X 0,Y 531.11,Z 220.827,A -85,B 0,C 180,E1 -4497.722,E2 -4497.722} C_VEL
LIN {X 0,Y 531.101,Z 220.825,A -85,B 0,C 180,E1 -4499.997,E2 -4499.997} C_VEL
LIN {X 0,Y 531.044,Z 220.832,A -85,B 0,C 180,E1 -4503.031,E2 -4503.031} C_VEL
LIN {X 0,Y 531.02,Z 220.837,A -85,B 0,C 180,E1 -4506.075,E2 -4506.075} C_VEL
LIN {X 0,Y 530.989,Z 220.837,A -85,B 0,C 180,E1 -4509.136,E2 -4509.136} C_VEL
LIN {X 0,Y 531.028,Z 220.839,A -85,B 0,C 180,E1 -4511.667,E2 -4511.667} C_VEL
LIN {X 0,Y 531,Z 220.836,A -85,B 0,C 180,E1 -4514.949,E2 -4514.949} C_VEL
LIN {X 0,Y 530.955,Z 220.845,A -85,B 0,C 180,E1 -4517.721,E2 -4517.721} C_VEL
LIN {X 0,Y 530.999,Z 220.844,A -85,B 0,C 180,E1 -4520.124,E2 -4520.124} C_VEL
LIN {X 0,Y 530.919,Z 220.849,A -85,B 0,C 180,E1 -4522.57,E2 -4522.57} C_VEL
LIN {X 0,Y 530.96,Z 220.84,A -85,B 0,C 180,E1 -4525.056,E2 -4525.056} C_VEL
LIN {X 0,Y 530.983,Z 220.839,A -85,B 0,C 180,E1 -4527.593,E2 -4527.593} C_VEL
LIN {X 0,Y 530.942,Z 220.849,A -85,B 0,C 180,E1 -4530.642,E2 -4530.642} C_VEL
LIN {X 0,Y 530.958,Z 220.842,A -85,B 0,C 180,E1 -4533.77,E2 -4533.77} C_VEL
LIN {X 0,Y 530.937,Z 220.852,A -85,B 0,C 180,E1 -4536.555,E2 -4536.555} C_VEL
LIN {X 0,Y 530.971,Z 220.841,A -85,B 0,C 180,E1 -4539.855,E2 -4539.855} C_VEL
LIN {X 0,Y 530.951,Z 220.849,A -85,B 0,C 180,E1 -4542.453,E2 -4542.453} C_VEL
LIN {X 0,Y 530.929,Z 220.847,A -85,B 0,C 180,E1 -4543.516,E2 -4543.516} C_VEL
LIN {X 0,Y 530.25,Z 220.933,A -85,B 0,C 180,E1 -4544.149,E2 -4544.149} C_VEL
LIN {X 0,Y 527.396,Z 221.292,A -85,B 0,C 180,E1 -4545.178,E2 -4545.178} C_VEL
LIN {X 0,Y 524.996,Z 221.593,A -85,B 0,C 180,E1 -4546.006,E2 -4546.006} C_VEL
LIN {X 0,Y 523.973,Z 221.72,A -85,B 0,C 180,E1 -4546.646,E2 -4546.646} C_VEL
LIN {X 0,Y 523.893,Z 221.73,A -85,B 0,C 180,E1 -4546.862,E2 -4546.862} C_VEL
LIN {X 0,Y 523.976,Z 221.965,A -85,B 0,C 180,E1 -4547.68,E2 -4547.68} C_VEL
LIN {X 0,Y 524.716,Z 227.972,A -85,B 0,C 180,E1 -4548.789,E2 -4548.789} C_VEL
LIN {X 0,Y 524.395,Z 243.169,A -85,B 0,C 180,E1 -4551.452,E2 -4551.452} C_VEL
LIN {X 0,Y 524.232,Z 257.225,A -85,B 0,C 180,E1 -4553.871,E2 -4553.871} C_VEL
LIN {X 0,Y 525.743,Z 266.12,A -85,B 0,C 180,E1 -4554.068,E2 -4554.068} C_VEL
LIN {X 0,Y 525.859,Z 279.996,A -85,B 0,C 180,E1 -4554.265,E2 -4554.265} C_VEL
LIN {X 0,Y 525.512,Z 364.809,A -85,B 0,C 180,E1 -4555.452,E2 -4555.452} C_VEL
LIN {X 0,Y 525.309,Z 378.62,A -85,B 0,C 180,E1 -4555.814,E2 -4555.814} C_VEL
LIN {X 0,Y 525.091,Z 391.153,A -85,B 0,C 180,E1 -4556.305,E2 -4556.305} C_VEL
LIN {X 0,Y 524.818,Z 402.908,A -85,B 0,C 180,E1 -4556.93,E2 -4556.93} C_VEL
LIN {X 0,Y 524.512,Z 414.295,A -85,B 0,C 180,E1 -4557.706,E2 -4557.706} C_VEL
LIN {X 0,Y 524.284,Z 423.488,A -85,B 0,C 180,E1 -4558.482,E2 -4558.482} C_VEL
LIN {X 0,Y 524.026,Z 432.133,A -85,B 0,C 180,E1 -4559.362,E2 -4559.362} C_VEL
LIN {X 0,Y 523.789,Z 441.293,A -85,B 0,C 180,E1 -4560.507,E2 -4560.507} C_VEL
LIN {X 0,Y 523.65,Z 449.302,A -85,B 0,C 180,E1 -4561.766,E2 -4561.766} C_VEL
LIN {X 0,Y 523.531,Z 454.804,A -85,B 0,C 180,E1 -4562.845,E2 -4562.845} C_VEL
LIN {X 0,Y 523.448,Z 459.84,A -85,B 0,C 180,E1 -4564.09,E2 -4564.09} C_VEL
LIN {X 0,Y 523.386,Z 463.784,A -85,B 0,C 180,E1 -4565.402,E2 -4565.402} C_VEL
LIN {X 0,Y 523.302,Z 465.604,A -85,B 0,C 180,E1 -4566.242,E2 -4566.242} C_VEL
LIN {X 0,Y 523.261,Z 466.96,A -85,B 0,C 180,E1 -4567.078,E2 -4567.078} C_VEL
LIN {X 0,Y 523.26,Z 467.828,A -85,B 0,C 180,E1 -4567.92,E2 -4567.92} C_VEL
LIN {X 0,Y 523.252,Z 468.205,A -85,B 0,C 180,E1 -4568.739,E2 -4568.739} C_VEL
LIN {X 0,Y 523.291,Z 467.895,A -85,B 0,C 180,E1 -4570.058,E2 -4570.058} C_VEL
LIN {X 0,Y 523.258,Z 466.687,A -85,B 0,C 180,E1 -4571.196,E2 -4571.196} C_VEL
LIN {X 0,Y 523.301,Z 464.331,A -85,B 0,C 180,E1 -4572.449,E2 -4572.449} C_VEL
LIN {X 0,Y 523.383,Z 461.09,A -85,B 0,C 180,E1 -4573.622,E2 -4573.622} C_VEL
LIN {X 0,Y 523.47,Z 456.479,A -85,B 0,C 180,E1 -4574.864,E2 -4574.864} C_VEL
LIN {X 0,Y 523.572,Z 450.971,A -85,B 0,C 180,E1 -4576.019,E2 -4576.019} C_VEL
LIN {X 0,Y 523.743,Z 443.877,A -85,B 0,C 180,E1 -4577.209,E2 -4577.209} C_VEL
LIN {X 0,Y 523.965,Z 434.988,A -85,B 0,C 180,E1 -4578.394,E2 -4578.394} C_VEL
LIN {X 0,Y 524.254,Z 424.895,A -85,B 0,C 180,E1 -4579.477,E2 -4579.477} C_VEL
LIN {X 0,Y 524.517,Z 414.6,A -85,B 0,C 180,E1 -4580.36,E2 -4580.36} C_VEL
LIN {X 0,Y 524.839,Z 403.163,A -85,B 0,C 180,E1 -4581.143,E2 -4581.143} C_VEL
LIN {X 0,Y 525.067,Z 391.405,A -85,B 0,C 180,E1 -4581.774,E2 -4581.774} C_VEL
LIN {X 0,Y 525.325,Z 378.909,A -85,B 0,C 180,E1 -4582.266,E2 -4582.266} C_VEL
LIN {X 0,Y 525.518,Z 366.303,A -85,B 0,C 180,E1 -4582.606,E2 -4582.606} C_VEL
LIN {X 0,Y 525.625,Z 342.183,A -85,B 0,C 180,E1 -4582.969,E2 -4582.969} C_VEL
LIN {X 0,Y 525.784,Z 266.192,A -85,B 0,C 180,E1 -4584.019,E2 -4584.019} C_VEL
LIN {X 0,Y 524.255,Z 257.525,A -85,B 0,C 180,E1 -4584.207,E2 -4584.207} C_VEL
LIN {X 0,Y 524.287,Z 253.826,A -85,B 0,C 180,E1 -4584.81,E2 -4584.81} C_VEL
LIN {X 0,Y 524.664,Z 237.85,A -85,B 0,C 180,E1 -4587.698,E2 -4587.698} C_VEL
LIN {X 0,Y 524.896,Z 227.358,A -85,B 0,C 180,E1 -4589.618,E2 -4589.618} C_VEL
LIN {X 0,Y 524.106,Z 221.794,A -85,B 0,C 180,E1 -4590.721,E2 -4590.721} C_VEL
LIN {X 0,Y 524.035,Z 221.712,A -85,B 0,C 180,E1 -4593.076,E2 -4593.076} C_VEL
LIN {X 0,Y 523.996,Z 221.71,A -85,B 0,C 180,E1 -4596.161,E2 -4596.161} C_VEL
LIN {X 0,Y 523.96,Z 221.712,A -85,B 0,C 180,E1 -4598.486,E2 -4598.486} C_VEL
LIN {X 0,Y 523.982,Z 221.717,A -85,B 0,C 180,E1 -4601.753,E2 -4601.753} C_VEL
LIN {X 0,Y 523.949,Z 221.714,A -85,B 0,C 180,E1 -4605.054,E2 -4605.054} C_VEL
LIN {X 0,Y 523.923,Z 221.724,A -85,B 0,C 180,E1 -4607.972,E2 -4607.972} C_VEL
LIN {X 0,Y 523.932,Z 221.718,A -85,B 0,C 180,E1 -4610.413,E2 -4610.413} C_VEL
LIN {X 0,Y 523.871,Z 221.723,A -85,B 0,C 180,E1 -4612.896,E2 -4612.896} C_VEL
LIN {X 0,Y 523.882,Z 221.723,A -85,B 0,C 180,E1 -4615.423,E2 -4615.423} C_VEL
LIN {X 0,Y 523.878,Z 221.73,A -85,B 0,C 180,E1 -4618.005,E2 -4618.005} C_VEL
LIN {X 0,Y 523.91,Z 221.72,A -85,B 0,C 180,E1 -4620.858,E2 -4620.858} C_VEL
LIN {X 0,Y 523.893,Z 221.722,A -85,B 0,C 180,E1 -4623.732,E2 -4623.732} C_VEL
LIN {X 0,Y 523.846,Z 221.737,A -85,B 0,C 180,E1 -4626.401,E2 -4626.401} C_VEL
LIN {X 0,Y 523.88,Z 221.724,A -85,B 0,C 180,E1 -4629.089,E2 -4629.089} C_VEL
LIN {X 0,Y 523.88,Z 221.725,A -85,B 0,C 180,E1 -4632.127,E2 -4632.127} C_VEL
LIN {X 0,Y 523.915,Z 221.719,A -85,B 0,C 180,E1 -4635.314,E2 -4635.314} C_VEL
LIN {X 0,Y 523.901,Z 221.728,A -85,B 0,C 180,E1 -4638.698,E2 -4638.698} C_VEL
LIN {X 0,Y 523.893,Z 221.72,A -85,B 0,C 180,E1 -4641.902,E2 -4641.902} C_VEL
LIN {X 0,Y 523.906,Z 221.727,A -85,B 0,C 180,E1 -4644.915,E2 -4644.915} C_VEL
LIN {X 0,Y 523.915,Z 221.719,A -85,B 0,C 180,E1 -4647.685,E2 -4647.685} C_VEL
LIN {X 0,Y 523.922,Z 221.719,A -85,B 0,C 180,E1 -4650.684,E2 -4650.684} C_VEL
LIN {X 0,Y 523.88,Z 221.725,A -85,B 0,C 180,E1 -4653.728,E2 -4653.728} C_VEL
LIN {X 0,Y 523.899,Z 221.72,A -85,B 0,C 180,E1 -4656.273,E2 -4656.273} C_VEL
LIN {X 0,Y 523.938,Z 221.716,A -85,B 0,C 180,E1 -4658.77,E2 -4658.77} C_VEL
LIN {X 0,Y 523.929,Z 221.721,A -85,B 0,C 180,E1 -4661.224,E2 -4661.224} C_VEL
LIN {X 0,Y 523.899,Z 221.73,A -85,B 0,C 180,E1 -4663.641,E2 -4663.641} C_VEL
LIN {X 0,Y 523.921,Z 221.722,A -85,B 0,C 180,E1 -4666.031,E2 -4666.031} C_VEL
LIN {X 0,Y 523.959,Z 221.714,A -85,B 0,C 180,E1 -4668.396,E2 -4668.396} C_VEL
LIN {X 0,Y 523.954,Z 221.717,A -85,B 0,C 180,E1 -4671.519,E2 -4671.519} C_VEL
LIN {X 0,Y 524.032,Z 221.704,A -85,B 0,C 180,E1 -4674.616,E2 -4674.616} C_VEL
LIN {X 0,Y 524.106,Z 221.698,A -85,B 0,C 180,E1 -4677.698,E2 -4677.698} C_VEL
LIN {X 0,Y 524.122,Z 221.694,A -85,B 0,C 180,E1 -4680.771,E2 -4680.771} C_VEL
LIN {X 0,Y 524.006,Z 221.707,A -85,B 0,C 180,E1 -4683.078,E2 -4683.078} C_VEL
LIN {X 0,Y 524.011,Z 221.712,A -85,B 0,C 180,E1 -4686.162,E2 -4686.162} C_VEL
LIN {X 0,Y 523.955,Z 221.713,A -85,B 0,C 180,E1 -4689.265,E2 -4689.265} C_VEL
LIN {X 0,Y 524.007,Z 221.706,A -85,B 0,C 180,E1 -4691.738,E2 -4691.738} C_VEL
LIN {X 0,Y 523.996,Z 221.711,A -85,B 0,C 180,E1 -4695.05,E2 -4695.05} C_VEL
LIN {X 0,Y 523.956,Z 221.713,A -85,B 0,C 180,E1 -4697.972,E2 -4697.972} C_VEL
LIN {X 0,Y 523.964,Z 221.715,A -85,B 0,C 180,E1 -4700.413,E2 -4700.413} C_VEL
LIN {X 0,Y 523.919,Z 221.728,A -85,B 0,C 180,E1 -4702.895,E2 -4702.895} C_VEL
LIN {X 0,Y 523.911,Z 221.721,A -85,B 0,C 180,E1 -4705.423,E2 -4705.423} C_VEL
LIN {X 0,Y 523.919,Z 221.717,A -85,B 0,C 180,E1 -4708.004,E2 -4708.004} C_VEL
LIN {X 0,Y 523.923,Z 221.722,A -85,B 0,C 180,E1 -4710.849,E2 -4710.849} C_VEL
LIN {X 0,Y 523.94,Z 221.717,A -85,B 0,C 180,E1 -4713.73,E2 -4713.73} C_VEL
LIN {X 0,Y 523.901,Z 221.719,A -85,B 0,C 180,E1 -4716.4,E2 -4716.4} C_VEL
LIN {X 0,Y 523.93,Z 221.72,A -85,B 0,C 180,E1 -4719.086,E2 -4719.086} C_VEL
LIN {X 0,Y 523.912,Z 221.72,A -85,B 0,C 180,E1 -4722.125,E2 -4722.125} C_VEL
LIN {X 0,Y 523.947,Z 221.719,A -85,B 0,C 180,E1 -4725.312,E2 -4725.312} C_VEL
LIN {X 0,Y 523.932,Z 221.715,A -85,B 0,C 180,E1 -4728.695,E2 -4728.695} C_VEL
LIN {X 0,Y 523.925,Z 221.726,A -85,B 0,C 180,E1 -4731.898,E2 -4731.898} C_VEL
LIN {X 0,Y 523.933,Z 221.715,A -85,B 0,C 180,E1 -4734.912,E2 -4734.912} C_VEL
